LIN {X 0,Y 256.114,Z 308.577,A -85,B 0,C 180,E1 -18381.118,E2 -18381.118} C_VEL
LIN {X 0,Y 256.131,Z 308.577,A -85,B 0,C 180,E1 -18385.131,E2 -18385.131} C_VEL
LIN {X 0,Y 256.077,Z 308.586,A -85,B 0,C 180,E1 -18388.587,E2 -18388.587} C_VEL
LIN {X 0,Y 256.039,Z 308.588,A -85,B 0,C 180,E1 -18391.704,E2 -18391.704} C_VEL
LIN {X 0,Y 256.048,Z 308.59,A -85,B 0,C 180,E1 -18395.197,E2 -18395.197} C_VEL
LIN {X 0,Y 256.081,Z 308.587,A -85,B 0,C 180,E1 -18397.274,E2 -18397.274} C_VEL
LIN {X 0,Y 256.021,Z 308.597,A -85,B 0,C 180,E1 -18401.209,E2 -18401.209} C_VEL
LIN {X 0,Y 256.015,Z 308.597,A -85,B 0,C 180,E1 -18405.539,E2 -18405.539} C_VEL
LIN {X 0,Y 256.03,Z 308.591,A -85,B 0,C 180,E1 -18408.801,E2 -18408.801} C_VEL
LIN {X 0,Y 256.103,Z 308.582,A -85,B 0,C 180,E1 -18412.871,E2 -18412.871} C_VEL
LIN {X 0,Y 256.142,Z 308.689,A -85,B 0,C 180,E1 -18414.221,E2 -18414.221} C_VEL
LIN {X 0,Y 259.197,Z 322.488,A -85,B 0,C 180,E1 -18418.563,E2 -18418.563} C_VEL
LIN {X 0,Y 261.811,Z 335.171,A -85,B 0,C 180,E1 -18422.354,E2 -18422.354} C_VEL
LIN {X 0,Y 261.634,Z 338.484,A -85,B 0,C 180,E1 -18423.267,E2 -18423.267} C_VEL
LIN {X 0,Y 260.691,Z 343.829,A -85,B 0,C 180,E1 -18424.698,E2 -18424.698} C_VEL
LIN {X 0,Y 262.51,Z 368.373,A -85,B 0,C 180,E1 -18425.713,E2 -18425.713} C_VEL
LIN {X 0,Y 263.496,Z 379.827,A -85,B 0,C 180,E1 -18426.176,E2 -18426.176} C_VEL
LIN {X 0,Y 261.358,Z 445.18,A -85,B 0,C 180,E1 -18428.461,E2 -18428.461} C_VEL
LIN {X 0,Y 260.854,Z 455.2,A -85,B 0,C 180,E1 -18428.987,E2 -18428.987} C_VEL
LIN {X 0,Y 260.148,Z 464.552,A -85,B 0,C 180,E1 -18429.651,E2 -18429.651} C_VEL
LIN {X 0,Y 259.438,Z 473.095,A -85,B 0,C 180,E1 -18430.419,E2 -18430.419} C_VEL
LIN {X 0,Y 258.581,Z 483.372,A -85,B 0,C 180,E1 -18431.587,E2 -18431.587} C_VEL
LIN {X 0,Y 257.769,Z 491.491,A -85,B 0,C 180,E1 -18432.709,E2 -18432.709} C_VEL
LIN {X 0,Y 256.852,Z 500.011,A -85,B 0,C 180,E1 -18434.125,E2 -18434.125} C_VEL
LIN {X 0,Y 256.062,Z 507.913,A -85,B 0,C 180,E1 -18435.704,E2 -18435.704} C_VEL
LIN {X 0,Y 255.478,Z 514.624,A -85,B 0,C 180,E1 -18437.291,E2 -18437.291} C_VEL
LIN {X 0,Y 254.899,Z 521.569,A -85,B 0,C 180,E1 -18439.279,E2 -18439.279} C_VEL
LIN {X 0,Y 254.571,Z 527.294,A -85,B 0,C 180,E1 -18441.271,E2 -18441.271} C_VEL
LIN {X 0,Y 254.459,Z 531.171,A -85,B 0,C 180,E1 -18442.864,E2 -18442.864} C_VEL
LIN {X 0,Y 254.426,Z 535.723,A -85,B 0,C 180,E1 -18445.25,E2 -18445.25} C_VEL
LIN {X 0,Y 254.312,Z 538.017,A -85,B 0,C 180,E1 -18446.835,E2 -18446.835} C_VEL
LIN {X 0,Y 254.579,Z 541.236,A -85,B 0,C 180,E1 -18450.003,E2 -18450.003} C_VEL
LIN {X 0,Y 254.198,Z 542.076,A -85,B 0,C 180,E1 -18451.587,E2 -18451.587} C_VEL
LIN {X 0,Y 254.17,Z 542.453,A -85,B 0,C 180,E1 -18453.173,E2 -18453.173} C_VEL
LIN {X 0,Y 254.083,Z 542.355,A -85,B 0,C 180,E1 -18455.282,E2 -18455.282} C_VEL
LIN {X 0,Y 254.247,Z 541.14,A -85,B 0,C 180,E1 -18457.947,E2 -18457.947} C_VEL
LIN {X 0,Y 254.567,Z 539.931,A -85,B 0,C 180,E1 -18459.537,E2 -18459.537} C_VEL
LIN {X 0,Y 255.342,Z 537.174,A -85,B 0,C 180,E1 -18461.915,E2 -18461.915} C_VEL
LIN {X 0,Y 256.555,Z 533.388,A -85,B 0,C 180,E1 -18464.275,E2 -18464.275} C_VEL
LIN {X 0,Y 258.302,Z 528.46,A -85,B 0,C 180,E1 -18466.602,E2 -18466.602} C_VEL
LIN {X 0,Y 260.277,Z 522.255,A -85,B 0,C 180,E1 -18468.908,E2 -18468.908} C_VEL
LIN {X 0,Y 262.432,Z 515.951,A -85,B 0,C 180,E1 -18470.785,E2 -18470.785} C_VEL
LIN {X 0,Y 265.001,Z 508.371,A -85,B 0,C 180,E1 -18472.617,E2 -18472.617} C_VEL
LIN {X 0,Y 267.173,Z 501.282,A -85,B 0,C 180,E1 -18474.063,E2 -18474.063} C_VEL
LIN {X 0,Y 269.672,Z 492.854,A -85,B 0,C 180,E1 -18475.469,E2 -18475.469} C_VEL
LIN {X 0,Y 271.95,Z 484.083,A -85,B 0,C 180,E1 -18476.681,E2 -18476.681} C_VEL
LIN {X 0,Y 274.07,Z 475.043,A -85,B 0,C 180,E1 -18477.696,E2 -18477.696} C_VEL
LIN {X 0,Y 276.051,Z 464.838,A -85,B 0,C 180,E1 -18478.617,E2 -18478.617} C_VEL
LIN {X 0,Y 277.859,Z 454.072,A -85,B 0,C 180,E1 -18479.345,E2 -18479.345} C_VEL
LIN {X 0,Y 279.297,Z 443.596,A -85,B 0,C 180,E1 -18479.852,E2 -18479.852} C_VEL
LIN {X 0,Y 283.965,Z 384.409,A -85,B 0,C 180,E1 -18481.995,E2 -18481.995} C_VEL
LIN {X 0,Y 282.949,Z 372.74,A -85,B 0,C 180,E1 -18482.847,E2 -18482.847} C_VEL
LIN {X 0,Y 281.976,Z 365.365,A -85,B 0,C 180,E1 -18483.5,E2 -18483.5} C_VEL
LIN {X 0,Y 277.7,Z 356.302,A -85,B 0,C 180,E1 -18485.107,E2 -18485.107} C_VEL
LIN {X 0,Y 274.684,Z 350.616,A -85,B 0,C 180,E1 -18486.34,E2 -18486.34} C_VEL
LIN {X 0,Y 272.069,Z 346.151,A -85,B 0,C 180,E1 -18487.432,E2 -18487.432} C_VEL
LIN {X 0,Y 269.572,Z 341.715,A -85,B 0,C 180,E1 -18488.685,E2 -18488.685} C_VEL
LIN {X 0,Y 267.905,Z 336.182,A -85,B 0,C 180,E1 -18491.747,E2 -18491.747} C_VEL
LIN {X 0,Y 266.481,Z 331.991,A -85,B 0,C 180,E1 -18494.597,E2 -18494.597} C_VEL
LIN {X 0,Y 265.102,Z 328.21,A -85,B 0,C 180,E1 -18497.925,E2 -18497.925} C_VEL
LIN {X 0,Y 263.893,Z 325.058,A -85,B 0,C 180,E1 -18502.228,E2 -18502.228} C_VEL
LIN {X 0,Y 263.574,Z 324.321,A -85,B 0,C 180,E1 -18504.084,E2 -18504.084} C_VEL
LIN {X 0,Y 263.401,Z 324.098,A -85,B 0,C 180,E1 -18508.626,E2 -18508.626} C_VEL
LIN {X 0,Y 263.901,Z 324.897,A -85,B 0,C 180,E1 -18511.497,E2 -18511.497} C_VEL
LIN {X 0,Y 264.788,Z 327.071,A -85,B 0,C 180,E1 -18514.871,E2 -18514.871} C_VEL
LIN {X 0,Y 265.88,Z 329.841,A -85,B 0,C 180,E1 -18517.685,E2 -18517.685} C_VEL
LIN {X 0,Y 267.613,Z 334.155,A -85,B 0,C 180,E1 -18520.976,E2 -18520.976} C_VEL
LIN {X 0,Y 269.587,Z 339.896,A -85,B 0,C 180,E1 -18524.309,E2 -18524.309} C_VEL
LIN {X 0,Y 273.841,Z 346.836,A -85,B 0,C 180,E1 -18526.245,E2 -18526.245} C_VEL
LIN {X 0,Y 277.114,Z 352.608,A -85,B 0,C 180,E1 -18527.621,E2 -18527.621} C_VEL
LIN {X 0,Y 280.442,Z 359.089,A -85,B 0,C 180,E1 -18528.924,E2 -18528.924} C_VEL
LIN {X 0,Y 281.228,Z 361.609,A -85,B 0,C 180,E1 -18529.283,E2 -18529.283} C_VEL
LIN {X 0,Y 283.281,Z 378.778,A -85,B 0,C 180,E1 -18530.847,E2 -18530.847} C_VEL
LIN {X 0,Y 283.529,Z 382.951,A -85,B 0,C 180,E1 -18531.149,E2 -18531.149} C_VEL
LIN {X 0,Y 278.983,Z 431.266,A -85,B 0,C 180,E1 -18533.128,E2 -18533.128} C_VEL
LIN {X 0,Y 277.298,Z 444.107,A -85,B 0,C 180,E1 -18533.908,E2 -18533.908} C_VEL
LIN {X 0,Y 275.485,Z 454.611,A -85,B 0,C 180,E1 -18534.828,E2 -18534.828} C_VEL
LIN {X 0,Y 273.394,Z 464.676,A -85,B 0,C 180,E1 -18535.947,E2 -18535.947} C_VEL
LIN {X 0,Y 271.189,Z 473.801,A -85,B 0,C 180,E1 -18537.216,E2 -18537.216} C_VEL
LIN {X 0,Y 268.712,Z 482.846,A -85,B 0,C 180,E1 -18538.782,E2 -18538.782} C_VEL
LIN {X 0,Y 265.9,Z 491.692,A -85,B 0,C 180,E1 -18540.758,E2 -18540.758} C_VEL
LIN {X 0,Y 263.929,Z 497.227,A -85,B 0,C 180,E1 -18542.29,E2 -18542.29} C_VEL
LIN {X 0,Y 262.192,Z 501.907,A -85,B 0,C 180,E1 -18543.843,E2 -18543.843} C_VEL
LIN {X 0,Y 260.615,Z 505.883,A -85,B 0,C 180,E1 -18545.459,E2 -18545.459} C_VEL
LIN {X 0,Y 258.633,Z 510.251,A -85,B 0,C 180,E1 -18547.81,E2 -18547.81} C_VEL
LIN {X 0,Y 257.521,Z 512.523,A -85,B 0,C 180,E1 -18549.425,E2 -18549.425} C_VEL
LIN {X 0,Y 256.563,Z 514.125,A -85,B 0,C 180,E1 -18551.056,E2 -18551.056} C_VEL
LIN {X 0,Y 255.746,Z 515.171,A -85,B 0,C 180,E1 -18552.701,E2 -18552.701} C_VEL
LIN {X 0,Y 254.877,Z 515.787,A -85,B 0,C 180,E1 -18555.192,E2 -18555.192} C_VEL
LIN {X 0,Y 254.291,Z 515.154,A -85,B 0,C 180,E1 -18557.7,E2 -18557.7} C_VEL
LIN {X 0,Y 254.076,Z 513.537,A -85,B 0,C 180,E1 -18559.875,E2 -18559.875} C_VEL
LIN {X 0,Y 254.058,Z 511.101,A -85,B 0,C 180,E1 -18561.93,E2 -18561.93} C_VEL
LIN {X 0,Y 254.346,Z 506.669,A -85,B 0,C 180,E1 -18564.487,E2 -18564.487} C_VEL
LIN {X 0,Y 254.594,Z 502.794,A -85,B 0,C 180,E1 -18566.212,E2 -18566.212} C_VEL
LIN {X 0,Y 255.028,Z 497.402,A -85,B 0,C 180,E1 -18568.138,E2 -18568.138} C_VEL
LIN {X 0,Y 255.458,Z 492.196,A -85,B 0,C 180,E1 -18569.684,E2 -18569.684} C_VEL
LIN {X 0,Y 256.07,Z 485.08,A -85,B 0,C 180,E1 -18571.432,E2 -18571.432} C_VEL
LIN {X 0,Y 256.763,Z 477.44,A -85,B 0,C 180,E1 -18572.983,E2 -18572.983} C_VEL
LIN {X 0,Y 257.589,Z 468.46,A -85,B 0,C 180,E1 -18574.482,E2 -18574.482} C_VEL
LIN {X 0,Y 258.507,Z 457.069,A -85,B 0,C 180,E1 -18576.003,E2 -18576.003} C_VEL
LIN {X 0,Y 259.295,Z 446.195,A -85,B 0,C 180,E1 -18577.091,E2 -18577.091} C_VEL
LIN {X 0,Y 259.852,Z 435.418,A -85,B 0,C 180,E1 -18577.913,E2 -18577.913} C_VEL
LIN {X 0,Y 260.388,Z 424.12,A -85,B 0,C 180,E1 -18578.524,E2 -18578.524} C_VEL
LIN {X 0,Y 262.234,Z 371.857,A -85,B 0,C 180,E1 -18580.561,E2 -18580.561} C_VEL
LIN {X 0,Y 258.762,Z 340.403,A -85,B 0,C 180,E1 -18582.011,E2 -18582.011} C_VEL
LIN {X 0,Y 260.138,Z 329.508,A -85,B 0,C 180,E1 -18585.379,E2 -18585.379} C_VEL
LIN {X 0,Y 258.66,Z 320.931,A -85,B 0,C 180,E1 -18588.266,E2 -18588.266} C_VEL
LIN {X 0,Y 256.154,Z 308.576,A -85,B 0,C 180,E1 -18592.672,E2 -18592.672} C_VEL
LIN {X 0,Y 256.068,Z 308.585,A -85,B 0,C 180,E1 -18596.707,E2 -18596.707} C_VEL
LIN {X 0,Y 256.044,Z 308.591,A -85,B 0,C 180,E1 -18600.391,E2 -18600.391} C_VEL
LIN {X 0,Y 256.069,Z 308.588,A -85,B 0,C 180,E1 -18603.951,E2 -18603.951} C_VEL
LIN {X 0,Y 256.062,Z 308.586,A -85,B 0,C 180,E1 -18607.402,E2 -18607.402} C_VEL
LIN {X 0,Y 256.134,Z 308.581,A -85,B 0,C 180,E1 -18610.774,E2 -18610.774} C_VEL
LIN {X 0,Y 256.236,Z 308.564,A -85,B 0,C 180,E1 -18614.079,E2 -18614.079} C_VEL
LIN {X 0,Y 256.293,Z 308.56,A -85,B 0,C 180,E1 -18618.931,E2 -18618.931} C_VEL
LIN {X 0,Y 256.473,Z 308.534,A -85,B 0,C 180,E1 -18622.123,E2 -18622.123} C_VEL
LIN {X 0,Y 256.447,Z 308.537,A -85,B 0,C 180,E1 -18626.855,E2 -18626.855} C_VEL
LIN {X 0,Y 256.698,Z 308.507,A -85,B 0,C 180,E1 -18628.428,E2 -18628.428} C_VEL
LIN {X 0,Y 256.697,Z 308.509,A -85,B 0,C 180,E1 -18631.566,E2 -18631.566} C_VEL
LIN {X 0,Y 256.455,Z 308.54,A -85,B 0,C 180,E1 -18636.289,E2 -18636.289} C_VEL
LIN {X 0,Y 256.428,Z 308.54,A -85,B 0,C 180,E1 -18639.461,E2 -18639.461} C_VEL
LIN {X 0,Y 256.231,Z 308.566,A -85,B 0,C 180,E1 -18644.287,E2 -18644.287} C_VEL
LIN {X 0,Y 256.16,Z 308.574,A -85,B 0,C 180,E1 -18647.56,E2 -18647.56} C_VEL
LIN {X 0,Y 256.117,Z 308.58,A -85,B 0,C 180,E1 -18651.093,E2 -18651.093} C_VEL
LIN {X 0,Y 256.125,Z 308.582,A -85,B 0,C 180,E1 -18655.106,E2 -18655.106} C_VEL
LIN {X 0,Y 256.042,Z 308.589,A -85,B 0,C 180,E1 -18659.602,E2 -18659.602} C_VEL
LIN {X 0,Y 256.053,Z 308.588,A -85,B 0,C 180,E1 -18663.287,E2 -18663.287} C_VEL
LIN {X 0,Y 256.095,Z 308.582,A -85,B 0,C 180,E1 -18667.263,E2 -18667.263} C_VEL
LIN {X 0,Y 256.035,Z 308.588,A -85,B 0,C 180,E1 -18671.198,E2 -18671.198} C_VEL
LIN {X 0,Y 256.019,Z 308.591,A -85,B 0,C 180,E1 -18675.529,E2 -18675.529} C_VEL
LIN {X 0,Y 256.026,Z 308.592,A -85,B 0,C 180,E1 -18678.79,E2 -18678.79} C_VEL
LIN {X 0,Y 256.099,Z 308.585,A -85,B 0,C 180,E1 -18682.861,E2 -18682.861} C_VEL
LIN {X 0,Y 256.039,Z 308.59,A -85,B 0,C 180,E1 -18686.702,E2 -18686.702} C_VEL
LIN {X 0,Y 256.082,Z 308.583,A -85,B 0,C 180,E1 -18690.395,E2 -18690.395} C_VEL
LIN {X 0,Y 256.136,Z 308.576,A -85,B 0,C 180,E1 -18694.867,E2 -18694.867} C_VEL
LIN {X 0,Y 256.087,Z 308.583,A -85,B 0,C 180,E1 -18699.097,E2 -18699.097} C_VEL
LIN {X 0,Y 256.19,Z 308.572,A -85,B 0,C 180,E1 -18704.077,E2 -18704.077} C_VEL
LIN {X 0,Y 256.251,Z 308.563,A -85,B 0,C 180,E1 -18708.931,E2 -18708.931} C_VEL
LIN {X 0,Y 256.469,Z 308.537,A -85,B 0,C 180,E1 -18712.124,E2 -18712.124} C_VEL
LIN {X 0,Y 256.464,Z 308.54,A -85,B 0,C 180,E1 -18716.857,E2 -18716.857} C_VEL
LIN {X 0,Y 256.713,Z 308.504,A -85,B 0,C 180,E1 -18719.999,E2 -18719.999} C_VEL
LIN {X 0,Y 256.453,Z 308.54,A -85,B 0,C 180,E1 -18723.141,E2 -18723.141} C_VEL
LIN {X 0,Y 256.468,Z 308.536,A -85,B 0,C 180,E1 -18727.874,E2 -18727.874} C_VEL
LIN {X 0,Y 256.233,Z 308.563,A -85,B 0,C 180,E1 -18731.3,E2 -18731.3} C_VEL
LIN {X 0,Y 256.224,Z 308.57,A -85,B 0,C 180,E1 -18735.919,E2 -18735.919} C_VEL
LIN {X 0,Y 256.128,Z 308.576,A -85,B 0,C 180,E1 -18738.13,E2 -18738.13} C_VEL
LIN {X 0,Y 255.453,Z 308.663,A -85,B 0,C 180,E1 -18739.44,E2 -18739.44} C_VEL
LIN {X 0,Y 252.641,Z 309.011,A -85,B 0,C 180,E1 -18741.579,E2 -18741.579} C_VEL
LIN {X 0,Y 250.245,Z 309.312,A -85,B 0,C 180,E1 -18743.318,E2 -18743.318} C_VEL
LIN {X 0,Y 249.191,Z 309.444,A -85,B 0,C 180,E1 -18744.666,E2 -18744.666} C_VEL
LIN {X 0,Y 249.091,Z 309.454,A -85,B 0,C 180,E1 -18745.123,E2 -18745.123} C_VEL
LIN {X 0,Y 249.019,Z 309.462,A -85,B 0,C 180,E1 -18748.983,E2 -18748.983} C_VEL
LIN {X 0,Y 248.994,Z 309.468,A -85,B 0,C 180,E1 -18752.43,E2 -18752.43} C_VEL
LIN {X 0,Y 248.996,Z 309.466,A -85,B 0,C 180,E1 -18756.35,E2 -18756.35} C_VEL
LIN {X 0,Y 248.961,Z 309.472,A -85,B 0,C 180,E1 -18760.486,E2 -18760.486} C_VEL
LIN {X 0,Y 248.97,Z 309.471,A -85,B 0,C 180,E1 -18762.794,E2 -18762.794} C_VEL
LIN {X 0,Y 248.984,Z 309.471,A -85,B 0,C 180,E1 -18767.366,E2 -18767.366} C_VEL
LIN {X 0,Y 249.002,Z 309.47,A -85,B 0,C 180,E1 -18771.624,E2 -18771.624} C_VEL
LIN {X 0,Y 249.091,Z 309.561,A -85,B 0,C 180,E1 -18773.797,E2 -18773.797} C_VEL
LIN {X 0,Y 252.249,Z 323.917,A -85,B 0,C 180,E1 -18778.434,E2 -18778.434} C_VEL
LIN {X 0,Y 254.682,Z 335.639,A -85,B 0,C 180,E1 -18782.03,E2 -18782.03} C_VEL
LIN {X 0,Y 254.729,Z 338.753,A -85,B 0,C 180,E1 -18782.926,E2 -18782.926} C_VEL
LIN {X 0,Y 253.753,Z 344.225,A -85,B 0,C 180,E1 -18784.369,E2 -18784.369} C_VEL
LIN {X 0,Y 255.793,Z 371.229,A -85,B 0,C 180,E1 -18785.501,E2 -18785.501} C_VEL
LIN {X 0,Y 256.565,Z 379.574,A -85,B 0,C 180,E1 -18785.853,E2 -18785.853} C_VEL
LIN {X 0,Y 254.365,Z 444.942,A -85,B 0,C 180,E1 -18788.212,E2 -18788.212} C_VEL
LIN {X 0,Y 253.843,Z 454.922,A -85,B 0,C 180,E1 -18788.751,E2 -18788.751} C_VEL
LIN {X 0,Y 253.09,Z 464.842,A -85,B 0,C 180,E1 -18789.483,E2 -18789.483} C_VEL
LIN {X 0,Y 252.375,Z 473.258,A -85,B 0,C 180,E1 -18790.272,E2 -18790.272} C_VEL
LIN {X 0,Y 251.502,Z 483.435,A -85,B 0,C 180,E1 -18791.472,E2 -18791.472} C_VEL
LIN {X 0,Y 250.668,Z 491.507,A -85,B 0,C 180,E1 -18792.627,E2 -18792.627} C_VEL
LIN {X 0,Y 249.746,Z 499.952,A -85,B 0,C 180,E1 -18794.081,E2 -18794.081} C_VEL
LIN {X 0,Y 248.973,Z 507.813,A -85,B 0,C 180,E1 -18795.705,E2 -18795.705} C_VEL
LIN {X 0,Y 248.37,Z 514.477,A -85,B 0,C 180,E1 -18797.337,E2 -18797.337} C_VEL
LIN {X 0,Y 247.802,Z 521.386,A -85,B 0,C 180,E1 -18799.381,E2 -18799.381} C_VEL
LIN {X 0,Y 247.534,Z 526.093,A -85,B 0,C 180,E1 -18801.02,E2 -18801.02} C_VEL
LIN {X 0,Y 247.369,Z 531.706,A -85,B 0,C 180,E1 -18803.479,E2 -18803.479} C_VEL
LIN {X 0,Y 247.376,Z 534.77,A -85,B 0,C 180,E1 -18805.115,E2 -18805.115} C_VEL
LIN {X 0,Y 247.282,Z 539.046,A -85,B 0,C 180,E1 -18808.375,E2 -18808.375} C_VEL
LIN {X 0,Y 247.524,Z 540.587,A -85,B 0,C 180,E1 -18810.003,E2 -18810.003} C_VEL
LIN {X 0,Y 247.097,Z 541.956,A -85,B 0,C 180,E1 -18813.264,E2 -18813.264} C_VEL
LIN {X 0,Y 246.987,Z 542.064,A -85,B 0,C 180,E1 -18815.185,E2 -18815.185} C_VEL
LIN {X 0,Y 247.186,Z 540.907,A -85,B 0,C 180,E1 -18818.175,E2 -18818.175} C_VEL
LIN {X 0,Y 247.546,Z 539.777,A -85,B 0,C 180,E1 -18819.81,E2 -18819.81} C_VEL
LIN {X 0,Y 248.355,Z 537.18,A -85,B 0,C 180,E1 -18822.256,E2 -18822.256} C_VEL
LIN {X 0,Y 249.684,Z 533.567,A -85,B 0,C 180,E1 -18824.676,E2 -18824.676} C_VEL
LIN {X 0,Y 251.515,Z 528.837,A -85,B 0,C 180,E1 -18827.063,E2 -18827.063} C_VEL
LIN {X 0,Y 253.59,Z 522.856,A -85,B 0,C 180,E1 -18829.426,E2 -18829.426} C_VEL
LIN {X 0,Y 256.338,Z 515.399,A -85,B 0,C 180,E1 -18831.725,E2 -18831.725} C_VEL
LIN {X 0,Y 259.098,Z 507.837,A -85,B 0,C 180,E1 -18833.585,E2 -18833.585} C_VEL
LIN {X 0,Y 261.414,Z 500.71,A -85,B 0,C 180,E1 -18835.052,E2 -18835.052} C_VEL
LIN {X 0,Y 264.071,Z 492.227,A -85,B 0,C 180,E1 -18836.474,E2 -18836.474} C_VEL
LIN {X 0,Y 266.497,Z 483.453,A -85,B 0,C 180,E1 -18837.698,E2 -18837.698} C_VEL
LIN {X 0,Y 268.708,Z 474.488,A -85,B 0,C 180,E1 -18838.725,E2 -18838.725} C_VEL
LIN {X 0,Y 270.801,Z 464.384,A -85,B 0,C 180,E1 -18839.652,E2 -18839.652} C_VEL
LIN {X 0,Y 272.745,Z 453.678,A -85,B 0,C 180,E1 -18840.377,E2 -18840.377} C_VEL
LIN {X 0,Y 274.212,Z 443.294,A -85,B 0,C 180,E1 -18840.887,E2 -18840.887} C_VEL
LIN {X 0,Y 279.082,Z 385.56,A -85,B 0,C 180,E1 -18843.024,E2 -18843.024} C_VEL
LIN {X 0,Y 278.145,Z 373.444,A -85,B 0,C 180,E1 -18843.959,E2 -18843.959} C_VEL
LIN {X 0,Y 277.492,Z 369.039,A -85,B 0,C 180,E1 -18844.387,E2 -18844.387} C_VEL
LIN {X 0,Y 273.757,Z 360.823,A -85,B 0,C 180,E1 -18845.922,E2 -18845.922} C_VEL
LIN {X 0,Y 271.155,Z 355.812,A -85,B 0,C 180,E1 -18847.037,E2 -18847.037} C_VEL
LIN {X 0,Y 268.946,Z 351.819,A -85,B 0,C 180,E1 -18848.051,E2 -18848.051} C_VEL
LIN {X 0,Y 265.932,Z 346.837,A -85,B 0,C 180,E1 -18849.507,E2 -18849.507} C_VEL
LIN {X 0,Y 262.807,Z 341.689,A -85,B 0,C 180,E1 -18851.279,E2 -18851.279} C_VEL
LIN {X 0,Y 261.347,Z 337.153,A -85,B 0,C 180,E1 -18854.36,E2 -18854.36} C_VEL
LIN {X 0,Y 260.116,Z 333.559,A -85,B 0,C 180,E1 -18857.511,E2 -18857.511} C_VEL
LIN {X 0,Y 258.911,Z 330.251,A -85,B 0,C 180,E1 -18861.921,E2 -18861.921} C_VEL
LIN {X 0,Y 258.743,Z 329.583,A -85,B 0,C 180,E1 -18863.305,E2 -18863.305} C_VEL
LIN {X 0,Y 258.326,Z 329.063,A -85,B 0,C 180,E1 -18867.496,E2 -18867.496} C_VEL
LIN {X 0,Y 258.727,Z 329.674,A -85,B 0,C 180,E1 -18870.73,E2 -18870.73} C_VEL
LIN {X 0,Y 259.348,Z 331.015,A -85,B 0,C 180,E1 -18873.409,E2 -18873.409} C_VEL
LIN {X 0,Y 260.395,Z 333.627,A -85,B 0,C 180,E1 -18876.58,E2 -18876.58} C_VEL
LIN {X 0,Y 261.852,Z 337.573,A -85,B 0,C 180,E1 -18879.942,E2 -18879.942} C_VEL
LIN {X 0,Y 262.835,Z 340.258,A -85,B 0,C 180,E1 -18881.692,E2 -18881.692} C_VEL
LIN {X 0,Y 267.268,Z 346.965,A -85,B 0,C 180,E1 -18884.071,E2 -18884.071} C_VEL
LIN {X 0,Y 270.636,Z 352.656,A -85,B 0,C 180,E1 -18885.703,E2 -18885.703} C_VEL
LIN {X 0,Y 274.341,Z 359.4,A -85,B 0,C 180,E1 -18887.318,E2 -18887.318} C_VEL
LIN {X 0,Y 276.669,Z 364.494,A -85,B 0,C 180,E1 -18888.326,E2 -18888.326} C_VEL
LIN {X 0,Y 278.512,Z 381.03,A -85,B 0,C 180,E1 -18889.884,E2 -18889.884} C_VEL
LIN {X 0,Y 278.564,Z 385.068,A -85,B 0,C 180,E1 -18890.159,E2 -18890.159} C_VEL
LIN {X 0,Y 273.873,Z 431.859,A -85,B 0,C 180,E1 -18892.119,E2 -18892.119} C_VEL
LIN {X 0,Y 272.197,Z 444.046,A -85,B 0,C 180,E1 -18892.863,E2 -18892.863} C_VEL
LIN {X 0,Y 270.197,Z 455.143,A -85,B 0,C 180,E1 -18893.841,E2 -18893.841} C_VEL
LIN {X 0,Y 268.114,Z 464.536,A -85,B 0,C 180,E1 -18894.897,E2 -18894.897} C_VEL
LIN {X 0,Y 266.027,Z 472.669,A -85,B 0,C 180,E1 -18896.024,E2 -18896.024} C_VEL
LIN {X 0,Y 263.793,Z 480.394,A -85,B 0,C 180,E1 -18897.329,E2 -18897.329} C_VEL
LIN {X 0,Y 261.635,Z 487.24,A -85,B 0,C 180,E1 -18898.714,E2 -18898.714} C_VEL
LIN {X 0,Y 259.753,Z 492.621,A -85,B 0,C 180,E1 -18900.001,E2 -18900.001} C_VEL
LIN {X 0,Y 257.69,Z 498.08,A -85,B 0,C 180,E1 -18901.564,E2 -18901.564} C_VEL
LIN {X 0,Y 255.803,Z 502.673,A -85,B 0,C 180,E1 -18903.151,E2 -18903.151} C_VEL
LIN {X 0,Y 253.946,Z 506.877,A -85,B 0,C 180,E1 -18904.955,E2 -18904.955} C_VEL
LIN {X 0,Y 251.991,Z 510.864,A -85,B 0,C 180,E1 -18907.211,E2 -18907.211} C_VEL
LIN {X 0,Y 249.934,Z 514.392,A -85,B 0,C 180,E1 -18910.218,E2 -18910.218} C_VEL
LIN {X 0,Y 248.487,Z 516.075,A -85,B 0,C 180,E1 -18913.078,E2 -18913.078} C_VEL
LIN {X 0,Y 247.749,Z 516.239,A -85,B 0,C 180,E1 -18915.323,E2 -18915.323} C_VEL
LIN {X 0,Y 247.117,Z 514.966,A -85,B 0,C 180,E1 -18918.231,E2 -18918.231} C_VEL
LIN {X 0,Y 246.984,Z 513.334,A -85,B 0,C 180,E1 -18920.118,E2 -18920.118} C_VEL
LIN {X 0,Y 246.97,Z 511.441,A -85,B 0,C 180,E1 -18921.713,E2 -18921.713} C_VEL
LIN {X 0,Y 247.197,Z 507.641,A -85,B 0,C 180,E1 -18924.012,E2 -18924.012} C_VEL
LIN {X 0,Y 247.494,Z 503.075,A -85,B 0,C 180,E1 -18926.114,E2 -18926.114} C_VEL
LIN {X 0,Y 247.937,Z 497.45,A -85,B 0,C 180,E1 -18928.169,E2 -18928.169} C_VEL
LIN {X 0,Y 248.35,Z 492.473,A -85,B 0,C 180,E1 -18929.686,E2 -18929.686} C_VEL
LIN {X 0,Y 248.987,Z 485.365,A -85,B 0,C 180,E1 -18931.48,E2 -18931.48} C_VEL
LIN {X 0,Y 249.684,Z 477.834,A -85,B 0,C 180,E1 -18933.05,E2 -18933.05} C_VEL
LIN {X 0,Y 250.379,Z 470.095,A -85,B 0,C 180,E1 -18934.396,E2 -18934.396} C_VEL
LIN {X 0,Y 251.048,Z 462.425,A -85,B 0,C 180,E1 -18935.514,E2 -18935.514} C_VEL
LIN {X 0,Y 251.709,Z 453.018,A -85,B 0,C 180,E1 -18936.643,E2 -18936.643} C_VEL
LIN {X 0,Y 252.518,Z 442.541,A -85,B 0,C 180,E1 -18937.631,E2 -18937.631} C_VEL
LIN {X 0,Y 253.17,Z 429.531,A -85,B 0,C 180,E1 -18938.511,E2 -18938.511} C_VEL
LIN {X 0,Y 254.256,Z 400.469,A -85,B 0,C 180,E1 -18939.734,E2 -18939.734} C_VEL
LIN {X 0,Y 255.242,Z 372.305,A -85,B 0,C 180,E1 -18940.859,E2 -18940.859} C_VEL
LIN {X 0,Y 251.813,Z 340.434,A -85,B 0,C 180,E1 -18942.391,E2 -18942.391} C_VEL
LIN {X 0,Y 253.127,Z 330.314,A -85,B 0,C 180,E1 -18945.595,E2 -18945.595} C_VEL
LIN {X 0,Y 251.53,Z 321.534,A -85,B 0,C 180,E1 -18948.63,E2 -18948.63} C_VEL
LIN {X 0,Y 249.184,Z 310,A -85,B 0,C 180,E1 -18952.816,E2 -18952.816} C_VEL
LIN {X 0,Y 249.098,Z 309.455,A -85,B 0,C 180,E1 -18953.127,E2 -18953.127} C_VEL
LIN {X 0,Y 249.034,Z 309.465,A -85,B 0,C 180,E1 -18957.849,E2 -18957.849} C_VEL
LIN {X 0,Y 249.038,Z 309.462,A -85,B 0,C 180,E1 -18961.33,E2 -18961.33} C_VEL
LIN {X 0,Y 249.059,Z 309.459,A -85,B 0,C 180,E1 -18964.958,E2 -18964.958} C_VEL
LIN {X 0,Y 249.056,Z 309.463,A -85,B 0,C 180,E1 -18968.627,E2 -18968.627} C_VEL
LIN {X 0,Y 249.164,Z 309.445,A -85,B 0,C 180,E1 -18973.615,E2 -18973.615} C_VEL
LIN {X 0,Y 249.192,Z 309.444,A -85,B 0,C 180,E1 -18976.958,E2 -18976.958} C_VEL
LIN {X 0,Y 249.389,Z 309.418,A -85,B 0,C 180,E1 -18980.52,E2 -18980.52} C_VEL
LIN {X 0,Y 249.43,Z 309.414,A -85,B 0,C 180,E1 -18983.526,E2 -18983.526} C_VEL
LIN {X 0,Y 249.659,Z 309.384,A -85,B 0,C 180,E1 -18988.384,E2 -18988.384} C_VEL
LIN {X 0,Y 249.658,Z 309.387,A -85,B 0,C 180,E1 -18991.61,E2 -18991.61} C_VEL
LIN {X 0,Y 249.429,Z 309.414,A -85,B 0,C 180,E1 -18996.467,E2 -18996.467} C_VEL
LIN {X 0,Y 249.345,Z 309.424,A -85,B 0,C 180,E1 -18999.732,E2 -18999.732} C_VEL
LIN {X 0,Y 249.17,Z 309.448,A -85,B 0,C 180,E1 -19004.701,E2 -19004.701} C_VEL
LIN {X 0,Y 249.092,Z 309.455,A -85,B 0,C 180,E1 -19008.076,E2 -19008.076} C_VEL
LIN {X 0,Y 249.041,Z 309.459,A -85,B 0,C 180,E1 -19011.517,E2 -19011.517} C_VEL
LIN {X 0,Y 249.077,Z 309.459,A -85,B 0,C 180,E1 -19015.454,E2 -19015.454} C_VEL
LIN {X 0,Y 249.025,Z 309.464,A -85,B 0,C 180,E1 -19018.967,E2 -19018.967} C_VEL
LIN {X 0,Y 249.015,Z 309.463,A -85,B 0,C 180,E1 -19022.421,E2 -19022.421} C_VEL
LIN {X 0,Y 249.012,Z 309.465,A -85,B 0,C 180,E1 -19026.34,E2 -19026.34} C_VEL
LIN {X 0,Y 248.974,Z 309.469,A -85,B 0,C 180,E1 -19030.475,E2 -19030.475} C_VEL
LIN {X 0,Y 248.982,Z 309.469,A -85,B 0,C 180,E1 -19032.784,E2 -19032.784} C_VEL
LIN {X 0,Y 248.984,Z 309.466,A -85,B 0,C 180,E1 -19037.355,E2 -19037.355} C_VEL
LIN {X 0,Y 249.015,Z 309.465,A -85,B 0,C 180,E1 -19042.196,E2 -19042.196} C_VEL
LIN {X 0,Y 249.015,Z 309.463,A -85,B 0,C 180,E1 -19045.634,E2 -19045.634} C_VEL
LIN {X 0,Y 249.021,Z 309.465,A -85,B 0,C 180,E1 -19049.468,E2 -19049.468} C_VEL
LIN {X 0,Y 249.037,Z 309.464,A -85,B 0,C 180,E1 -19053.157,E2 -19053.157} C_VEL
LIN {X 0,Y 249.022,Z 309.46,A -85,B 0,C 180,E1 -19056.726,E2 -19056.726} C_VEL
LIN {X 0,Y 249.009,Z 309.466,A -85,B 0,C 180,E1 -19060.202,E2 -19060.202} C_VEL
LIN {X 0,Y 249.122,Z 309.452,A -85,B 0,C 180,E1 -19063.613,E2 -19063.613} C_VEL
LIN {X 0,Y 249.194,Z 309.443,A -85,B 0,C 180,E1 -19068.613,E2 -19068.613} C_VEL
LIN {X 0,Y 249.407,Z 309.416,A -85,B 0,C 180,E1 -19071.9,E2 -19071.9} C_VEL
LIN {X 0,Y 249.257,Z 309.434,A -85,B 0,C 180,E1 -19075.147,E2 -19075.147} C_VEL
LIN {X 0,Y 249.636,Z 309.388,A -85,B 0,C 180,E1 -19078.386,E2 -19078.386} C_VEL
LIN {X 0,Y 249.632,Z 309.386,A -85,B 0,C 180,E1 -19081.612,E2 -19081.612} C_VEL
LIN {X 0,Y 249.407,Z 309.415,A -85,B 0,C 180,E1 -19086.471,E2 -19086.471} C_VEL
LIN {X 0,Y 249.304,Z 309.429,A -85,B 0,C 180,E1 -19089.737,E2 -19089.737} C_VEL
LIN {X 0,Y 249.145,Z 309.447,A -85,B 0,C 180,E1 -19094.706,E2 -19094.706} C_VEL
LIN {X 0,Y 249.089,Z 309.457,A -85,B 0,C 180,E1 -19098.102,E2 -19098.102} C_VEL
LIN {X 0,Y 249.047,Z 309.458,A -85,B 0,C 180,E1 -19101.521,E2 -19101.521} C_VEL
LIN {X 0,Y 249.091,Z 309.454,A -85,B 0,C 180,E1 -19105.123,E2 -19105.123} C_VEL
LIN {X 0,Y 248.364,Z 309.549,A -85,B 0,C 180,E1 -19106.472,E2 -19106.472} C_VEL
LIN {X 0,Y 245.434,Z 309.911,A -85,B 0,C 180,E1 -19108.67,E2 -19108.67} C_VEL
LIN {X 0,Y 243,Z 310.213,A -85,B 0,C 180,E1 -19110.46,E2 -19110.46} C_VEL
LIN {X 0,Y 241.997,Z 310.337,A -85,B 0,C 180,E1 -19111.85,E2 -19111.85} C_VEL
LIN {X 0,Y 241.937,Z 310.346,A -85,B 0,C 180,E1 -19112.321,E2 -19112.321} C_VEL
LIN {X 0,Y 241.948,Z 310.344,A -85,B 0,C 180,E1 -19115.591,E2 -19115.591} C_VEL
LIN {X 0,Y 241.917,Z 310.35,A -85,B 0,C 180,E1 -19119.726,E2 -19119.726} C_VEL
LIN {X 0,Y 241.891,Z 310.352,A -85,B 0,C 180,E1 -19124.21,E2 -19124.21} C_VEL
LIN {X 0,Y 241.909,Z 310.352,A -85,B 0,C 180,E1 -19128.081,E2 -19128.081} C_VEL
LIN {X 0,Y 241.974,Z 310.344,A -85,B 0,C 180,E1 -19132.424,E2 -19132.424} C_VEL
LIN {X 0,Y 242.042,Z 310.45,A -85,B 0,C 180,E1 -19133.357,E2 -19133.357} C_VEL
LIN {X 0,Y 244.685,Z 322.589,A -85,B 0,C 180,E1 -19137.423,E2 -19137.423} C_VEL
LIN {X 0,Y 247.169,Z 334.123,A -85,B 0,C 180,E1 -19141.101,E2 -19141.101} C_VEL
LIN {X 0,Y 247.801,Z 337.695,A -85,B 0,C 180,E1 -19142.201,E2 -19142.201} C_VEL
LIN {X 0,Y 247.244,Z 341.902,A -85,B 0,C 180,E1 -19143.41,E2 -19143.41} C_VEL
LIN {X 0,Y 246.837,Z 344.096,A -85,B 0,C 180,E1 -19143.989,E2 -19143.989} C_VEL
LIN {X 0,Y 248.625,Z 369.376,A -85,B 0,C 180,E1 -19145.074,E2 -19145.074} C_VEL
LIN {X 0,Y 249.577,Z 380.376,A -85,B 0,C 180,E1 -19145.549,E2 -19145.549} C_VEL
LIN {X 0,Y 247.389,Z 444.693,A -85,B 0,C 180,E1 -19147.949,E2 -19147.949} C_VEL
LIN {X 0,Y 246.846,Z 454.629,A -85,B 0,C 180,E1 -19148.502,E2 -19148.502} C_VEL
LIN {X 0,Y 246.127,Z 463.928,A -85,B 0,C 180,E1 -19149.203,E2 -19149.203} C_VEL
LIN {X 0,Y 245.323,Z 473.354,A -85,B 0,C 180,E1 -19150.117,E2 -19150.117} C_VEL
LIN {X 0,Y 244.558,Z 481.929,A -85,B 0,C 180,E1 -19151.143,E2 -19151.143} C_VEL
LIN {X 0,Y 243.637,Z 491.002,A -85,B 0,C 180,E1 -19152.469,E2 -19152.469} C_VEL
LIN {X 0,Y 242.66,Z 499.803,A -85,B 0,C 180,E1 -19154.035,E2 -19154.035} C_VEL
LIN {X 0,Y 241.87,Z 507.61,A -85,B 0,C 180,E1 -19155.706,E2 -19155.706} C_VEL
LIN {X 0,Y 241.291,Z 514.24,A -85,B 0,C 180,E1 -19157.387,E2 -19157.387} C_VEL
LIN {X 0,Y 240.735,Z 521.11,A -85,B 0,C 180,E1 -19159.491,E2 -19159.491} C_VEL
LIN {X 0,Y 240.41,Z 526.758,A -85,B 0,C 180,E1 -19161.599,E2 -19161.599} C_VEL
LIN {X 0,Y 240.315,Z 531.694,A -85,B 0,C 180,E1 -19163.887,E2 -19163.887} C_VEL
LIN {X 0,Y 240.26,Z 535.039,A -85,B 0,C 180,E1 -19165.81,E2 -19165.81} C_VEL
LIN {X 0,Y 240.21,Z 538.263,A -85,B 0,C 180,E1 -19168.327,E2 -19168.327} C_VEL
LIN {X 0,Y 240.469,Z 539.844,A -85,B 0,C 180,E1 -19170.003,E2 -19170.003} C_VEL
LIN {X 0,Y 240.026,Z 541.459,A -85,B 0,C 180,E1 -19173.36,E2 -19173.36} C_VEL
LIN {X 0,Y 239.909,Z 541.634,A -85,B 0,C 180,E1 -19175.13,E2 -19175.13} C_VEL
LIN {X 0,Y 240.145,Z 540.7,A -85,B 0,C 180,E1 -19178.417,E2 -19178.417} C_VEL
LIN {X 0,Y 240.511,Z 539.572,A -85,B 0,C 180,E1 -19180.1,E2 -19180.1} C_VEL
LIN {X 0,Y 241.756,Z 536.13,A -85,B 0,C 180,E1 -19183.45,E2 -19183.45} C_VEL
LIN {X 0,Y 243.427,Z 532.311,A -85,B 0,C 180,E1 -19185.921,E2 -19185.921} C_VEL
LIN {X 0,Y 245.446,Z 527.384,A -85,B 0,C 180,E1 -19188.361,E2 -19188.361} C_VEL
LIN {X 0,Y 247.784,Z 521.421,A -85,B 0,C 180,E1 -19190.68,E2 -19190.68} C_VEL
LIN {X 0,Y 250.362,Z 514.89,A -85,B 0,C 180,E1 -19192.706,E2 -19192.706} C_VEL
LIN {X 0,Y 253.236,Z 507.32,A -85,B 0,C 180,E1 -19194.602,E2 -19194.602} C_VEL
LIN {X 0,Y 255.78,Z 500.237,A -85,B 0,C 180,E1 -19196.081,E2 -19196.081} C_VEL
LIN {X 0,Y 258.579,Z 491.84,A -85,B 0,C 180,E1 -19197.52,E2 -19197.52} C_VEL
LIN {X 0,Y 261.132,Z 483.11,A -85,B 0,C 180,E1 -19198.756,E2 -19198.756} C_VEL
LIN {X 0,Y 263.459,Z 474.138,A -85,B 0,C 180,E1 -19199.791,E2 -19199.791} C_VEL
LIN {X 0,Y 265.696,Z 464.005,A -85,B 0,C 180,E1 -19200.72,E2 -19200.72} C_VEL
LIN {X 0,Y 267.716,Z 453.345,A -85,B 0,C 180,E1 -19201.45,E2 -19201.45} C_VEL
LIN {X 0,Y 269.262,Z 443.113,A -85,B 0,C 180,E1 -19201.962,E2 -19201.962} C_VEL
LIN {X 0,Y 274.383,Z 386.982,A -85,B 0,C 180,E1 -19204.085,E2 -19204.085} C_VEL
LIN {X 0,Y 273.543,Z 375.524,A -85,B 0,C 180,E1 -19205.012,E2 -19205.012} C_VEL
LIN {X 0,Y 273.158,Z 372.747,A -85,B 0,C 180,E1 -19205.301,E2 -19205.301} C_VEL
LIN {X 0,Y 269.928,Z 365.493,A -85,B 0,C 180,E1 -19206.734,E2 -19206.734} C_VEL
LIN {X 0,Y 266.484,Z 358.478,A -85,B 0,C 180,E1 -19208.382,E2 -19208.382} C_VEL
LIN {X 0,Y 262.9,Z 352.452,A -85,B 0,C 180,E1 -19210.212,E2 -19210.212} C_VEL
LIN {X 0,Y 259.689,Z 347.231,A -85,B 0,C 180,E1 -19212.09,E2 -19212.09} C_VEL
LIN {X 0,Y 255.94,Z 341.51,A -85,B 0,C 180,E1 -19214.763,E2 -19214.763} C_VEL
LIN {X 0,Y 254.724,Z 337.927,A -85,B 0,C 180,E1 -19218.153,E2 -19218.153} C_VEL
LIN {X 0,Y 253.801,Z 335.016,A -85,B 0,C 180,E1 -19222.469,E2 -19222.469} C_VEL
LIN {X 0,Y 253.525,Z 334.347,A -85,B 0,C 180,E1 -19224.4,E2 -19224.4} C_VEL
LIN {X 0,Y 253.477,Z 334.338,A -85,B 0,C 180,E1 -19229.259,E2 -19229.259} C_VEL
LIN {X 0,Y 254.037,Z 335.373,A -85,B 0,C 180,E1 -19232.283,E2 -19232.283} C_VEL
LIN {X 0,Y 254.883,Z 337.721,A -85,B 0,C 180,E1 -19235.57,E2 -19235.57} C_VEL
LIN {X 0,Y 255.994,Z 340.539,A -85,B 0,C 180,E1 -19238.246,E2 -19238.246} C_VEL
LIN {X 0,Y 260.594,Z 346.995,A -85,B 0,C 180,E1 -19241.373,E2 -19241.373} C_VEL
LIN {X 0,Y 264.407,Z 352.987,A -85,B 0,C 180,E1 -19243.547,E2 -19243.547} C_VEL
LIN {X 0,Y 267.512,Z 358.457,A -85,B 0,C 180,E1 -19245.132,E2 -19245.132} C_VEL
LIN {X 0,Y 271.141,Z 365.412,A -85,B 0,C 180,E1 -19246.827,E2 -19246.827} C_VEL
LIN {X 0,Y 272.44,Z 368.518,A -85,B 0,C 180,E1 -19247.439,E2 -19247.439} C_VEL
LIN {X 0,Y 273.864,Z 383.787,A -85,B 0,C 180,E1 -19248.914,E2 -19248.914} C_VEL
LIN {X 0,Y 273.862,Z 386.129,A -85,B 0,C 180,E1 -19249.073,E2 -19249.073} C_VEL
LIN {X 0,Y 269.001,Z 432.053,A -85,B 0,C 180,E1 -19251.029,E2 -19251.029} C_VEL
LIN {X 0,Y 267.217,Z 444.169,A -85,B 0,C 180,E1 -19251.779,E2 -19251.779} C_VEL
LIN {X 0,Y 265.067,Z 455.278,A -85,B 0,C 180,E1 -19252.766,E2 -19252.766} C_VEL
LIN {X 0,Y 262.808,Z 464.928,A -85,B 0,C 180,E1 -19253.86,E2 -19253.86} C_VEL
LIN {X 0,Y 260.545,Z 473.37,A -85,B 0,C 180,E1 -19255.051,E2 -19255.051} C_VEL
LIN {X 0,Y 258.295,Z 480.679,A -85,B 0,C 180,E1 -19256.296,E2 -19256.296} C_VEL
LIN {X 0,Y 256.087,Z 487.234,A -85,B 0,C 180,E1 -19257.642,E2 -19257.642} C_VEL
LIN {X 0,Y 253.474,Z 494.09,A -85,B 0,C 180,E1 -19259.347,E2 -19259.347} C_VEL
LIN {X 0,Y 250.936,Z 500.149,A -85,B 0,C 180,E1 -19261.204,E2 -19261.204} C_VEL
LIN {X 0,Y 249.447,Z 503.482,A -85,B 0,C 180,E1 -19262.423,E2 -19262.423} C_VEL
LIN {X 0,Y 247.684,Z 507.251,A -85,B 0,C 180,E1 -19264.069,E2 -19264.069} C_VEL
LIN {X 0,Y 245.382,Z 511.521,A -85,B 0,C 180,E1 -19266.579,E2 -19266.579} C_VEL
LIN {X 0,Y 244.076,Z 513.694,A -85,B 0,C 180,E1 -19268.279,E2 -19268.279} C_VEL
LIN {X 0,Y 242.819,Z 515.453,A -85,B 0,C 180,E1 -19270.252,E2 -19270.252} C_VEL
LIN {X 0,Y 241.997,Z 516.212,A -85,B 0,C 180,E1 -19271.73,E2 -19271.73} C_VEL
LIN {X 0,Y 241.221,Z 516.647,A -85,B 0,C 180,E1 -19273.479,E2 -19273.479} C_VEL
LIN {X 0,Y 240.623,Z 516.501,A -85,B 0,C 180,E1 -19275.461,E2 -19275.461} C_VEL
LIN {X 0,Y 240.242,Z 515.967,A -85,B 0,C 180,E1 -19277.011,E2 -19277.011} C_VEL
LIN {X 0,Y 239.951,Z 514.708,A -85,B 0,C 180,E1 -19278.796,E2 -19278.796} C_VEL
LIN {X 0,Y 239.861,Z 511.774,A -85,B 0,C 180,E1 -19281.486,E2 -19281.486} C_VEL
LIN {X 0,Y 240.118,Z 507.247,A -85,B 0,C 180,E1 -19284.191,E2 -19284.191} C_VEL
LIN {X 0,Y 240.388,Z 503.329,A -85,B 0,C 180,E1 -19286.012,E2 -19286.012} C_VEL
LIN {X 0,Y 240.743,Z 498.509,A -85,B 0,C 180,E1 -19287.846,E2 -19287.846} C_VEL
LIN {X 0,Y 241.253,Z 492.646,A -85,B 0,C 180,E1 -19289.686,E2 -19289.686} C_VEL
LIN {X 0,Y 241.9,Z 485.502,A -85,B 0,C 180,E1 -19291.532,E2 -19291.532} C_VEL
LIN {X 0,Y 242.629,Z 477.79,A -85,B 0,C 180,E1 -19293.181,E2 -19293.181} C_VEL
LIN {X 0,Y 243.455,Z 468.812,A -85,B 0,C 180,E1 -19294.761,E2 -19294.761} C_VEL
LIN {X 0,Y 244.442,Z 457.162,A -85,B 0,C 180,E1 -19296.389,E2 -19296.389} C_VEL
LIN {X 0,Y 245.239,Z 446.479,A -85,B 0,C 180,E1 -19297.517,E2 -19297.517} C_VEL
LIN {X 0,Y 245.797,Z 436.109,A -85,B 0,C 180,E1 -19298.357,E2 -19298.357} C_VEL
LIN {X 0,Y 246.366,Z 424.765,A -85,B 0,C 180,E1 -19299.011,E2 -19299.011} C_VEL
LIN {X 0,Y 248.285,Z 372.957,A -85,B 0,C 180,E1 -19301.164,E2 -19301.164} C_VEL
LIN {X 0,Y 244.884,Z 340.469,A -85,B 0,C 180,E1 -19302.765,E2 -19302.765} C_VEL
LIN {X 0,Y 246.058,Z 331.852,A -85,B 0,C 180,E1 -19305.568,E2 -19305.568} C_VEL
LIN {X 0,Y 245.462,Z 327.393,A -85,B 0,C 180,E1 -19307.123,E2 -19307.123} C_VEL
LIN {X 0,Y 243.206,Z 315.955,A -85,B 0,C 180,E1 -19311.283,E2 -19311.283} C_VEL
LIN {X 0,Y 242.036,Z 310.335,A -85,B 0,C 180,E1 -19313.47,E2 -19313.47} C_VEL
LIN {X 0,Y 241.99,Z 310.34,A -85,B 0,C 180,E1 -19317.378,E2 -19317.378} C_VEL
LIN {X 0,Y 241.974,Z 310.342,A -85,B 0,C 180,E1 -19320.616,E2 -19320.616} C_VEL
LIN {X 0,Y 242,Z 310.343,A -85,B 0,C 180,E1 -19324.197,E2 -19324.197} C_VEL
LIN {X 0,Y 241.991,Z 310.343,A -85,B 0,C 180,E1 -19328.337,E2 -19328.337} C_VEL
LIN {X 0,Y 242.12,Z 310.323,A -85,B 0,C 180,E1 -19333.317,E2 -19333.317} C_VEL
LIN {X 0,Y 242.171,Z 310.315,A -85,B 0,C 180,E1 -19338.277,E2 -19338.277} C_VEL
LIN {X 0,Y 242.377,Z 310.292,A -85,B 0,C 180,E1 -19341.661,E2 -19341.661} C_VEL
LIN {X 0,Y 242.401,Z 310.291,A -85,B 0,C 180,E1 -19343.338,E2 -19343.338} C_VEL
LIN {X 0,Y 242.618,Z 310.261,A -85,B 0,C 180,E1 -19348.337,E2 -19348.337} C_VEL
LIN {X 0,Y 242.618,Z 310.264,A -85,B 0,C 180,E1 -19351.656,E2 -19351.656} C_VEL
LIN {X 0,Y 242.402,Z 310.288,A -85,B 0,C 180,E1 -19356.656,E2 -19356.656} C_VEL
LIN {X 0,Y 242.268,Z 310.307,A -85,B 0,C 180,E1 -19360.019,E2 -19360.019} C_VEL
LIN {X 0,Y 242.125,Z 310.323,A -85,B 0,C 180,E1 -19365.138,E2 -19365.138} C_VEL
LIN {X 0,Y 242.028,Z 310.338,A -85,B 0,C 180,E1 -19368.622,E2 -19368.622} C_VEL
LIN {X 0,Y 241.982,Z 310.337,A -85,B 0,C 180,E1 -19372.177,E2 -19372.177} C_VEL
LIN {X 0,Y 242.025,Z 310.335,A -85,B 0,C 180,E1 -19375.815,E2 -19375.815} C_VEL
LIN {X 0,Y 241.958,Z 310.343,A -85,B 0,C 180,E1 -19379.583,E2 -19379.583} C_VEL
LIN {X 0,Y 241.967,Z 310.344,A -85,B 0,C 180,E1 -19383.487,E2 -19383.487} C_VEL
LIN {X 0,Y 241.968,Z 310.343,A -85,B 0,C 180,E1 -19387.577,E2 -19387.577} C_VEL
LIN {X 0,Y 241.911,Z 310.35,A -85,B 0,C 180,E1 -19391.918,E2 -19391.918} C_VEL
LIN {X 0,Y 241.901,Z 310.351,A -85,B 0,C 180,E1 -19396.569,E2 -19396.569} C_VEL
LIN {X 0,Y 241.969,Z 310.341,A -85,B 0,C 180,E1 -19401.636,E2 -19401.636} C_VEL
LIN {X 0,Y 241.952,Z 310.345,A -85,B 0,C 180,E1 -19404.482,E2 -19404.482} C_VEL
LIN {X 0,Y 241.945,Z 310.343,A -85,B 0,C 180,E1 -19408.474,E2 -19408.474} C_VEL
LIN {X 0,Y 241.974,Z 310.341,A -85,B 0,C 180,E1 -19412.307,E2 -19412.307} C_VEL
LIN {X 0,Y 242.004,Z 310.336,A -85,B 0,C 180,E1 -19416.009,E2 -19416.009} C_VEL
LIN {X 0,Y 241.95,Z 310.347,A -85,B 0,C 180,E1 -19419.599,E2 -19419.599} C_VEL
LIN {X 0,Y 242.079,Z 310.328,A -85,B 0,C 180,E1 -19423.315,E2 -19423.315} C_VEL
LIN {X 0,Y 242.128,Z 310.326,A -85,B 0,C 180,E1 -19428.276,E2 -19428.276} C_VEL
LIN {X 0,Y 242.354,Z 310.293,A -85,B 0,C 180,E1 -19431.662,E2 -19431.662} C_VEL
LIN {X 0,Y 242.217,Z 310.311,A -85,B 0,C 180,E1 -19435.005,E2 -19435.005} C_VEL
LIN {X 0,Y 242.597,Z 310.265,A -85,B 0,C 180,E1 -19438.339,E2 -19438.339} C_VEL
LIN {X 0,Y 242.593,Z 310.262,A -85,B 0,C 180,E1 -19441.659,E2 -19441.659} C_VEL
LIN {X 0,Y 242.378,Z 310.291,A -85,B 0,C 180,E1 -19446.659,E2 -19446.659} C_VEL
LIN {X 0,Y 242.228,Z 310.309,A -85,B 0,C 180,E1 -19450.024,E2 -19450.024} C_VEL
LIN {X 0,Y 242.102,Z 310.325,A -85,B 0,C 180,E1 -19455.144,E2 -19455.144} C_VEL
LIN {X 0,Y 242.028,Z 310.333,A -85,B 0,C 180,E1 -19458.627,E2 -19458.627} C_VEL
LIN {X 0,Y 241.969,Z 310.344,A -85,B 0,C 180,E1 -19462.183,E2 -19462.183} C_VEL
LIN {X 0,Y 242.016,Z 310.337,A -85,B 0,C 180,E1 -19465.832,E2 -19465.832} C_VEL
LIN {X 0,Y 241.942,Z 310.342,A -85,B 0,C 180,E1 -19469.591,E2 -19469.591} C_VEL
LIN {X 0,Y 241.937,Z 310.346,A -85,B 0,C 180,E1 -19472.321,E2 -19472.321} C_VEL
LIN {X 0,Y 241.323,Z 310.429,A -85,B 0,C 180,E1 -19473.711,E2 -19473.711} C_VEL
LIN {X 0,Y 238.481,Z 310.785,A -85,B 0,C 180,E1 -19475.976,E2 -19475.976} C_VEL
LIN {X 0,Y 236.015,Z 311.088,A -85,B 0,C 180,E1 -19477.821,E2 -19477.821} C_VEL
LIN {X 0,Y 234.929,Z 311.223,A -85,B 0,C 180,E1 -19479.254,E2 -19479.254} C_VEL
LIN {X 0,Y 234.828,Z 311.231,A -85,B 0,C 180,E1 -19479.741,E2 -19479.741} C_VEL
LIN {X 0,Y 234.856,Z 311.229,A -85,B 0,C 180,E1 -19484.105,E2 -19484.105} C_VEL
LIN {X 0,Y 234.858,Z 311.229,A -85,B 0,C 180,E1 -19488.836,E2 -19488.836} C_VEL
LIN {X 0,Y 234.994,Z 311.391,A -85,B 0,C 180,E1 -19492.937,E2 -19492.937} C_VEL
LIN {X 0,Y 237.438,Z 322.584,A -85,B 0,C 180,E1 -19496.806,E2 -19496.806} C_VEL
LIN {X 0,Y 240.062,Z 334.792,A -85,B 0,C 180,E1 -19500.82,E2 -19500.82} C_VEL
LIN {X 0,Y 240.803,Z 339.038,A -85,B 0,C 180,E1 -19502.169,E2 -19502.169} C_VEL
LIN {X 0,Y 239.939,Z 343.991,A -85,B 0,C 180,E1 -19503.593,E2 -19503.593} C_VEL
LIN {X 0,Y 241.538,Z 368.486,A -85,B 0,C 180,E1 -19504.677,E2 -19504.677} C_VEL
LIN {X 0,Y 242.608,Z 380.591,A -85,B 0,C 180,E1 -19505.219,E2 -19505.219} C_VEL
LIN {X 0,Y 240.355,Z 444.757,A -85,B 0,C 180,E1 -19507.721,E2 -19507.721} C_VEL
LIN {X 0,Y 239.821,Z 454.541,A -85,B 0,C 180,E1 -19508.292,E2 -19508.292} C_VEL
LIN {X 0,Y 239.091,Z 463.773,A -85,B 0,C 180,E1 -19509.013,E2 -19509.013} C_VEL
LIN {X 0,Y 238.262,Z 473.151,A -85,B 0,C 180,E1 -19509.952,E2 -19509.952} C_VEL
LIN {X 0,Y 237.484,Z 481.699,A -85,B 0,C 180,E1 -19511.008,E2 -19511.008} C_VEL
LIN {X 0,Y 236.492,Z 491.287,A -85,B 0,C 180,E1 -19512.466,E2 -19512.466} C_VEL
LIN {X 0,Y 235.583,Z 499.545,A -85,B 0,C 180,E1 -19513.987,E2 -19513.987} C_VEL
LIN {X 0,Y 234.772,Z 507.332,A -85,B 0,C 180,E1 -19515.707,E2 -19515.707} C_VEL
LIN {X 0,Y 234.189,Z 513.947,A -85,B 0,C 180,E1 -19517.438,E2 -19517.438} C_VEL
LIN {X 0,Y 233.644,Z 520.803,A -85,B 0,C 180,E1 -19519.607,E2 -19519.607} C_VEL
LIN {X 0,Y 233.377,Z 525.461,A -85,B 0,C 180,E1 -19521.344,E2 -19521.344} C_VEL
LIN {X 0,Y 233.256,Z 530.875,A -85,B 0,C 180,E1 -19523.866,E2 -19523.866} C_VEL
LIN {X 0,Y 233.212,Z 534.063,A -85,B 0,C 180,E1 -19525.683,E2 -19525.683} C_VEL
LIN {X 0,Y 233.139,Z 537.467,A -85,B 0,C 180,E1 -19528.276,E2 -19528.276} C_VEL
LIN {X 0,Y 233.413,Z 539.057,A -85,B 0,C 180,E1 -19530.003,E2 -19530.003} C_VEL
LIN {X 0,Y 232.956,Z 540.938,A -85,B 0,C 180,E1 -19533.462,E2 -19533.462} C_VEL
LIN {X 0,Y 232.878,Z 540.955,A -85,B 0,C 180,E1 -19536.936,E2 -19536.936} C_VEL
LIN {X 0,Y 233.092,Z 540.448,A -85,B 0,C 180,E1 -19538.673,E2 -19538.673} C_VEL
LIN {X 0,Y 234.08,Z 537.965,A -85,B 0,C 180,E1 -19542.135,E2 -19542.135} C_VEL
LIN {X 0,Y 235.364,Z 535.041,A -85,B 0,C 180,E1 -19544.705,E2 -19544.705} C_VEL
LIN {X 0,Y 237.279,Z 531.065,A -85,B 0,C 180,E1 -19547.231,E2 -19547.231} C_VEL
LIN {X 0,Y 239.46,Z 525.943,A -85,B 0,C 180,E1 -19549.727,E2 -19549.727} C_VEL
LIN {X 0,Y 241.799,Z 520.714,A -85,B 0,C 180,E1 -19551.753,E2 -19551.753} C_VEL
LIN {X 0,Y 244.47,Z 514.484,A -85,B 0,C 180,E1 -19553.734,E2 -19553.734} C_VEL
LIN {X 0,Y 247.517,Z 506.989,A -85,B 0,C 180,E1 -19555.659,E2 -19555.659} C_VEL
LIN {X 0,Y 250.594,Z 498.899,A -85,B 0,C 180,E1 -19557.339,E2 -19557.339} C_VEL
LIN {X 0,Y 253.572,Z 490.305,A -85,B 0,C 180,E1 -19558.788,E2 -19558.788} C_VEL
LIN {X 0,Y 256.281,Z 481.418,A -85,B 0,C 180,E1 -19560.031,E2 -19560.031} C_VEL
LIN {X 0,Y 258.74,Z 472.293,A -85,B 0,C 180,E1 -19561.07,E2 -19561.07} C_VEL
LIN {X 0,Y 260.927,Z 462.985,A -85,B 0,C 180,E1 -19561.911,E2 -19561.911} C_VEL
LIN {X 0,Y 262.941,Z 452.94,A -85,B 0,C 180,E1 -19562.598,E2 -19562.598} C_VEL
LIN {X 0,Y 264.532,Z 442.725,A -85,B 0,C 180,E1 -19563.113,E2 -19563.113} C_VEL
LIN {X 0,Y 269.813,Z 388.313,A -85,B 0,C 180,E1 -19565.212,E2 -19565.212} C_VEL
LIN {X 0,Y 269.262,Z 378.411,A -85,B 0,C 180,E1 -19566.038,E2 -19566.038} C_VEL
LIN {X 0,Y 268.866,Z 376.182,A -85,B 0,C 180,E1 -19566.309,E2 -19566.309} C_VEL
LIN {X 0,Y 265.427,Z 368.313,A -85,B 0,C 180,E1 -19567.983,E2 -19567.983} C_VEL
LIN {X 0,Y 262.273,Z 362.274,A -85,B 0,C 180,E1 -19569.597,E2 -19569.597} C_VEL
LIN {X 0,Y 260.112,Z 358.305,A -85,B 0,C 180,E1 -19570.842,E2 -19570.842} C_VEL
LIN {X 0,Y 257.071,Z 353.178,A -85,B 0,C 180,E1 -19572.744,E2 -19572.744} C_VEL
LIN {X 0,Y 253.487,Z 347.661,A -85,B 0,C 180,E1 -19575.428,E2 -19575.428} C_VEL
LIN {X 0,Y 249.806,Z 342.573,A -85,B 0,C 180,E1 -19579.207,E2 -19579.207} C_VEL
LIN {X 0,Y 248.999,Z 341.053,A -85,B 0,C 180,E1 -19580.672,E2 -19580.672} C_VEL
LIN {X 0,Y 248.668,Z 339.557,A -85,B 0,C 180,E1 -19583.594,E2 -19583.594} C_VEL
LIN {X 0,Y 248.391,Z 339.236,A -85,B 0,C 180,E1 -19588.081,E2 -19588.081} C_VEL
LIN {X 0,Y 248.809,Z 340.019,A -85,B 0,C 180,E1 -19591.303,E2 -19591.303} C_VEL
LIN {X 0,Y 249.337,Z 340.997,A -85,B 0,C 180,E1 -19592.987,E2 -19592.987} C_VEL
LIN {X 0,Y 252.812,Z 345.697,A -85,B 0,C 180,E1 -19596.898,E2 -19596.898} C_VEL
LIN {X 0,Y 254.409,Z 347.928,A -85,B 0,C 180,E1 -19598.264,E2 -19598.264} C_VEL
LIN {X 0,Y 257.986,Z 353.143,A -85,B 0,C 180,E1 -19600.827,E2 -19600.827} C_VEL
LIN {X 0,Y 261.486,Z 358.855,A -85,B 0,C 180,E1 -19602.952,E2 -19602.952} C_VEL
LIN {X 0,Y 264.692,Z 364.759,A -85,B 0,C 180,E1 -19604.682,E2 -19604.682} C_VEL
LIN {X 0,Y 268.109,Z 371.974,A -85,B 0,C 180,E1 -19606.415,E2 -19606.415} C_VEL
LIN {X 0,Y 269.074,Z 381.041,A -85,B 0,C 180,E1 -19607.394,E2 -19607.394} C_VEL
LIN {X 0,Y 269.362,Z 387.033,A -85,B 0,C 180,E1 -19607.926,E2 -19607.926} C_VEL
LIN {X 0,Y 264.191,Z 433.035,A -85,B 0,C 180,E1 -19609.931,E2 -19609.931} C_VEL
LIN {X 0,Y 262.186,Z 445.729,A -85,B 0,C 180,E1 -19610.746,E2 -19610.746} C_VEL
LIN {X 0,Y 259.726,Z 457.399,A -85,B 0,C 180,E1 -19611.834,E2 -19611.834} C_VEL
LIN {X 0,Y 257.709,Z 465.32,A -85,B 0,C 180,E1 -19612.755,E2 -19612.755} C_VEL
LIN {X 0,Y 255.363,Z 473.481,A -85,B 0,C 180,E1 -19613.924,E2 -19613.924} C_VEL
LIN {X 0,Y 252.551,Z 481.969,A -85,B 0,C 180,E1 -19615.412,E2 -19615.412} C_VEL
LIN {X 0,Y 250.21,Z 488.419,A -85,B 0,C 180,E1 -19616.78,E2 -19616.78} C_VEL
LIN {X 0,Y 247.672,Z 494.671,A -85,B 0,C 180,E1 -19618.375,E2 -19618.375} C_VEL
LIN {X 0,Y 245.326,Z 499.919,A -85,B 0,C 180,E1 -19620.001,E2 -19620.001} C_VEL
LIN {X 0,Y 243.172,Z 504.327,A -85,B 0,C 180,E1 -19621.657,E2 -19621.657} C_VEL
LIN {X 0,Y 240.496,Z 509.337,A -85,B 0,C 180,E1 -19624.084,E2 -19624.084} C_VEL
LIN {X 0,Y 238.815,Z 512.202,A -85,B 0,C 180,E1 -19625.913,E2 -19625.913} C_VEL
LIN {X 0,Y 236.756,Z 515.099,A -85,B 0,C 180,E1 -19628.536,E2 -19628.536} C_VEL
LIN {X 0,Y 235.671,Z 516.316,A -85,B 0,C 180,E1 -19630.308,E2 -19630.308} C_VEL
LIN {X 0,Y 234.723,Z 517.044,A -85,B 0,C 180,E1 -19632.099,E2 -19632.099} C_VEL
LIN {X 0,Y 233.99,Z 517.19,A -85,B 0,C 180,E1 -19633.904,E2 -19633.904} C_VEL
LIN {X 0,Y 233.454,Z 516.712,A -85,B 0,C 180,E1 -19635.721,E2 -19635.721} C_VEL
LIN {X 0,Y 233.025,Z 515.716,A -85,B 0,C 180,E1 -19637.555,E2 -19637.555} C_VEL
LIN {X 0,Y 232.79,Z 512.822,A -85,B 0,C 180,E1 -19640.632,E2 -19640.632} C_VEL
LIN {X 0,Y 232.873,Z 509.25,A -85,B 0,C 180,E1 -19643.101,E2 -19643.101} C_VEL
LIN {X 0,Y 233.187,Z 505.017,A -85,B 0,C 180,E1 -19645.293,E2 -19645.293} C_VEL
LIN {X 0,Y 233.644,Z 498.722,A -85,B 0,C 180,E1 -19647.791,E2 -19647.791} C_VEL
LIN {X 0,Y 234.21,Z 492.027,A -85,B 0,C 180,E1 -19649.909,E2 -19649.909} C_VEL
LIN {X 0,Y 234.907,Z 484.62,A -85,B 0,C 180,E1 -19651.825,E2 -19651.825} C_VEL
LIN {X 0,Y 235.623,Z 476.845,A -85,B 0,C 180,E1 -19653.487,E2 -19653.487} C_VEL
LIN {X 0,Y 236.669,Z 465.847,A -85,B 0,C 180,E1 -19655.386,E2 -19655.386} C_VEL
LIN {X 0,Y 237.432,Z 456.316,A -85,B 0,C 180,E1 -19656.669,E2 -19656.669} C_VEL
LIN {X 0,Y 238.164,Z 447.132,A -85,B 0,C 180,E1 -19657.663,E2 -19657.663} C_VEL
LIN {X 0,Y 238.786,Z 436.616,A -85,B 0,C 180,E1 -19658.547,E2 -19658.547} C_VEL
LIN {X 0,Y 239.324,Z 425.482,A -85,B 0,C 180,E1 -19659.22,E2 -19659.22} C_VEL
LIN {X 0,Y 241.281,Z 373.338,A -85,B 0,C 180,E1 -19661.487,E2 -19661.487} C_VEL
LIN {X 0,Y 237.928,Z 340.664,A -85,B 0,C 180,E1 -19663.123,E2 -19663.123} C_VEL
LIN {X 0,Y 239.051,Z 332.286,A -85,B 0,C 180,E1 -19665.908,E2 -19665.908} C_VEL
LIN {X 0,Y 237.321,Z 322.87,A -85,B 0,C 180,E1 -19669.345,E2 -19669.345} C_VEL
LIN {X 0,Y 235.231,Z 312.507,A -85,B 0,C 180,E1 -19673.306,E2 -19673.306} C_VEL
LIN {X 0,Y 234.988,Z 311.213,A -85,B 0,C 180,E1 -19673.855,E2 -19673.855} C_VEL
LIN {X 0,Y 234.955,Z 311.217,A -85,B 0,C 180,E1 -19677.424,E2 -19677.424} C_VEL
LIN {X 0,Y 234.894,Z 311.224,A -85,B 0,C 180,E1 -19681.398,E2 -19681.398} C_VEL
LIN {X 0,Y 234.918,Z 311.221,A -85,B 0,C 180,E1 -19685.238,E2 -19685.238} C_VEL
LIN {X 0,Y 234.945,Z 311.218,A -85,B 0,C 180,E1 -19688.962,E2 -19688.962} C_VEL
LIN {X 0,Y 235.061,Z 311.204,A -85,B 0,C 180,E1 -19693.092,E2 -19693.092} C_VEL
LIN {X 0,Y 235.103,Z 311.196,A -85,B 0,C 180,E1 -19697.919,E2 -19697.919} C_VEL
LIN {X 0,Y 235.317,Z 311.173,A -85,B 0,C 180,E1 -19701.409,E2 -19701.409} C_VEL
LIN {X 0,Y 235.352,Z 311.168,A -85,B 0,C 180,E1 -19703.137,E2 -19703.137} C_VEL
LIN {X 0,Y 235.577,Z 311.138,A -85,B 0,C 180,E1 -19708.287,E2 -19708.287} C_VEL
LIN {X 0,Y 235.577,Z 311.141,A -85,B 0,C 180,E1 -19711.706,E2 -19711.706} C_VEL
LIN {X 0,Y 235.354,Z 311.166,A -85,B 0,C 180,E1 -19716.856,E2 -19716.856} C_VEL
LIN {X 0,Y 235.215,Z 311.186,A -85,B 0,C 180,E1 -19720.323,E2 -19720.323} C_VEL
LIN {X 0,Y 235.073,Z 311.2,A -85,B 0,C 180,E1 -19725.604,E2 -19725.604} C_VEL
LIN {X 0,Y 234.966,Z 311.215,A -85,B 0,C 180,E1 -19729.203,E2 -19729.203} C_VEL
LIN {X 0,Y 234.932,Z 311.219,A -85,B 0,C 180,E1 -19732.88,E2 -19732.88} C_VEL
LIN {X 0,Y 234.937,Z 311.218,A -85,B 0,C 180,E1 -19736.655,E2 -19736.655} C_VEL
LIN {X 0,Y 234.888,Z 311.22,A -85,B 0,C 180,E1 -19740.567,E2 -19740.567} C_VEL
LIN {X 0,Y 234.912,Z 311.221,A -85,B 0,C 180,E1 -19744.633,E2 -19744.633} C_VEL
LIN {X 0,Y 234.896,Z 311.22,A -85,B 0,C 180,E1 -19748.929,E2 -19748.929} C_VEL
LIN {X 0,Y 234.858,Z 311.228,A -85,B 0,C 180,E1 -19753.482,E2 -19753.482} C_VEL
LIN {X 0,Y 234.854,Z 311.23,A -85,B 0,C 180,E1 -19756.505,E2 -19756.505} C_VEL
LIN {X 0,Y 234.895,Z 311.224,A -85,B 0,C 180,E1 -19761.073,E2 -19761.073} C_VEL
LIN {X 0,Y 234.898,Z 311.222,A -85,B 0,C 180,E1 -19765.355,E2 -19765.355} C_VEL
LIN {X 0,Y 234.902,Z 311.224,A -85,B 0,C 180,E1 -19769.427,E2 -19769.427} C_VEL
LIN {X 0,Y 234.964,Z 311.215,A -85,B 0,C 180,E1 -19773.79,E2 -19773.79} C_VEL
LIN {X 0,Y 234.92,Z 311.221,A -85,B 0,C 180,E1 -19778.011,E2 -19778.011} C_VEL
LIN {X 0,Y 235.02,Z 311.206,A -85,B 0,C 180,E1 -19783.091,E2 -19783.091} C_VEL
LIN {X 0,Y 235.06,Z 311.204,A -85,B 0,C 180,E1 -19787.918,E2 -19787.918} C_VEL
LIN {X 0,Y 235.282,Z 311.174,A -85,B 0,C 180,E1 -19791.41,E2 -19791.41} C_VEL
LIN {X 0,Y 235.329,Z 311.166,A -85,B 0,C 180,E1 -19793.138,E2 -19793.138} C_VEL
LIN {X 0,Y 235.557,Z 311.141,A -85,B 0,C 180,E1 -19798.289,E2 -19798.289} C_VEL
LIN {X 0,Y 235.552,Z 311.139,A -85,B 0,C 180,E1 -19801.709,E2 -19801.709} C_VEL
LIN {X 0,Y 235.329,Z 311.17,A -85,B 0,C 180,E1 -19806.86,E2 -19806.86} C_VEL
LIN {X 0,Y 235.174,Z 311.186,A -85,B 0,C 180,E1 -19810.328,E2 -19810.328} C_VEL
LIN {X 0,Y 235.056,Z 311.206,A -85,B 0,C 180,E1 -19815.609,E2 -19815.609} C_VEL
LIN {X 0,Y 234.966,Z 311.213,A -85,B 0,C 180,E1 -19819.208,E2 -19819.208} C_VEL
LIN {X 0,Y 234.916,Z 311.22,A -85,B 0,C 180,E1 -19822.886,E2 -19822.886} C_VEL
LIN {X 0,Y 234.922,Z 311.221,A -85,B 0,C 180,E1 -19826.662,E2 -19826.662} C_VEL
LIN {X 0,Y 234.869,Z 311.227,A -85,B 0,C 180,E1 -19830.576,E2 -19830.576} C_VEL
LIN {X 0,Y 234.894,Z 311.226,A -85,B 0,C 180,E1 -19834.643,E2 -19834.643} C_VEL
LIN {X 0,Y 234.884,Z 311.228,A -85,B 0,C 180,E1 -19838.939,E2 -19838.939} C_VEL
LIN {X 0,Y 234.828,Z 311.231,A -85,B 0,C 180,E1 -19839.741,E2 -19839.741} C_VEL
LIN {X 0,Y 234.129,Z 311.323,A -85,B 0,C 180,E1 -19841.173,E2 -19841.173} C_VEL
LIN {X 0,Y 231.281,Z 311.677,A -85,B 0,C 180,E1 -19843.51,E2 -19843.51} C_VEL
LIN {X 0,Y 228.884,Z 311.976,A -85,B 0,C 180,E1 -19845.415,E2 -19845.415} C_VEL
LIN {X 0,Y 227.862,Z 312.102,A -85,B 0,C 180,E1 -19846.893,E2 -19846.893} C_VEL
LIN {X 0,Y 227.78,Z 312.112,A -85,B 0,C 180,E1 -19847.394,E2 -19847.394} C_VEL
LIN {X 0,Y 227.942,Z 312.254,A -85,B 0,C 180,E1 -19852.469,E2 -19852.469} C_VEL
LIN {X 0,Y 230.549,Z 324.21,A -85,B 0,C 180,E1 -19856.73,E2 -19856.73} C_VEL
LIN {X 0,Y 233.187,Z 336.596,A -85,B 0,C 180,E1 -19860.928,E2 -19860.928} C_VEL
LIN {X 0,Y 233.701,Z 340.613,A -85,B 0,C 180,E1 -19862.224,E2 -19862.224} C_VEL
LIN {X 0,Y 233.04,Z 343.855,A -85,B 0,C 180,E1 -19863.2,E2 -19863.2} C_VEL
LIN {X 0,Y 234.339,Z 365.701,A -85,B 0,C 180,E1 -19864.2,E2 -19864.2} C_VEL
LIN {X 0,Y 235.621,Z 381.704,A -85,B 0,C 180,E1 -19864.934,E2 -19864.934} C_VEL
LIN {X 0,Y 233.326,Z 444.734,A -85,B 0,C 180,E1 -19867.48,E2 -19867.48} C_VEL
LIN {X 0,Y 232.736,Z 455.172,A -85,B 0,C 180,E1 -19868.121,E2 -19868.121} C_VEL
LIN {X 0,Y 231.957,Z 464.747,A -85,B 0,C 180,E1 -19868.918,E2 -19868.918} C_VEL
LIN {X 0,Y 231.212,Z 472.951,A -85,B 0,C 180,E1 -19869.778,E2 -19869.778} C_VEL
LIN {X 0,Y 230.358,Z 482.046,A -85,B 0,C 180,E1 -19870.949,E2 -19870.949} C_VEL
LIN {X 0,Y 229.389,Z 491.197,A -85,B 0,C 180,E1 -19872.395,E2 -19872.395} C_VEL
LIN {X 0,Y 228.509,Z 499.288,A -85,B 0,C 180,E1 -19873.936,E2 -19873.936} C_VEL
LIN {X 0,Y 227.672,Z 507.055,A -85,B 0,C 180,E1 -19875.708,E2 -19875.708} C_VEL
LIN {X 0,Y 227.094,Z 513.656,A -85,B 0,C 180,E1 -19877.494,E2 -19877.494} C_VEL
LIN {X 0,Y 226.569,Z 520.49,A -85,B 0,C 180,E1 -19879.73,E2 -19879.73} C_VEL
LIN {X 0,Y 226.282,Z 526.09,A -85,B 0,C 180,E1 -19881.97,E2 -19881.97} C_VEL
LIN {X 0,Y 226.225,Z 531.415,A -85,B 0,C 180,E1 -19884.656,E2 -19884.656} C_VEL
LIN {X 0,Y 226.096,Z 535.393,A -85,B 0,C 180,E1 -19887.331,E2 -19887.331} C_VEL
LIN {X 0,Y 226.358,Z 538.23,A -85,B 0,C 180,E1 -19890.004,E2 -19890.004} C_VEL
LIN {X 0,Y 225.91,Z 539.486,A -85,B 0,C 180,E1 -19891.786,E2 -19891.786} C_VEL
LIN {X 0,Y 225.888,Z 540.315,A -85,B 0,C 180,E1 -19893.571,E2 -19893.571} C_VEL
LIN {X 0,Y 225.806,Z 540.599,A -85,B 0,C 180,E1 -19897.155,E2 -19897.155} C_VEL
LIN {X 0,Y 226.059,Z 540.107,A -85,B 0,C 180,E1 -19898.945,E2 -19898.945} C_VEL
LIN {X 0,Y 227.096,Z 537.952,A -85,B 0,C 180,E1 -19902.514,E2 -19902.514} C_VEL
LIN {X 0,Y 228.493,Z 535.197,A -85,B 0,C 180,E1 -19905.158,E2 -19905.158} C_VEL
LIN {X 0,Y 230.522,Z 531.395,A -85,B 0,C 180,E1 -19907.752,E2 -19907.752} C_VEL
LIN {X 0,Y 233.195,Z 525.653,A -85,B 0,C 180,E1 -19910.694,E2 -19910.694} C_VEL
LIN {X 0,Y 235.769,Z 520.376,A -85,B 0,C 180,E1 -19912.801,E2 -19912.801} C_VEL
LIN {X 0,Y 238.717,Z 514.139,A -85,B 0,C 180,E1 -19914.806,E2 -19914.806} C_VEL
LIN {X 0,Y 241.901,Z 506.656,A -85,B 0,C 180,E1 -19916.765,E2 -19916.765} C_VEL
LIN {X 0,Y 244.83,Z 499.654,A -85,B 0,C 180,E1 -19918.272,E2 -19918.272} C_VEL
LIN {X 0,Y 247.938,Z 491.383,A -85,B 0,C 180,E1 -19919.74,E2 -19919.74} C_VEL
LIN {X 0,Y 250.774,Z 482.812,A -85,B 0,C 180,E1 -19920.995,E2 -19920.995} C_VEL
LIN {X 0,Y 253.771,Z 472.348,A -85,B 0,C 180,E1 -19922.216,E2 -19922.216} C_VEL
LIN {X 0,Y 256.073,Z 463.122,A -85,B 0,C 180,E1 -19923.057,E2 -19923.057} C_VEL
LIN {X 0,Y 258.419,Z 451.928,A -85,B 0,C 180,E1 -19923.826,E2 -19923.826} C_VEL
LIN {X 0,Y 260.073,Z 441.698,A -85,B 0,C 180,E1 -19924.34,E2 -19924.34} C_VEL
LIN {X 0,Y 265.478,Z 389.551,A -85,B 0,C 180,E1 -19926.391,E2 -19926.391} C_VEL
LIN {X 0,Y 265.018,Z 380.622,A -85,B 0,C 180,E1 -19927.171,E2 -19927.171} C_VEL
LIN {X 0,Y 261.882,Z 373.12,A -85,B 0,C 180,E1 -19928.847,E2 -19928.847} C_VEL
LIN {X 0,Y 259.376,Z 368.016,A -85,B 0,C 180,E1 -19930.254,E2 -19930.254} C_VEL
LIN {X 0,Y 257.069,Z 363.657,A -85,B 0,C 180,E1 -19931.663,E2 -19931.663} C_VEL
LIN {X 0,Y 254.638,Z 359.375,A -85,B 0,C 180,E1 -19933.323,E2 -19933.323} C_VEL
LIN {X 0,Y 251.284,Z 353.9,A -85,B 0,C 180,E1 -19936.046,E2 -19936.046} C_VEL
LIN {X 0,Y 247.816,Z 348.819,A -85,B 0,C 180,E1 -19939.969,E2 -19939.969} C_VEL
LIN {X 0,Y 246.733,Z 347.161,A -85,B 0,C 180,E1 -19941.909,E2 -19941.909} C_VEL
LIN {X 0,Y 245.92,Z 346.06,A -85,B 0,C 180,E1 -19944.137,E2 -19944.137} C_VEL
LIN {X 0,Y 245.624,Z 345.791,A -85,B 0,C 180,E1 -19947.069,E2 -19947.069} C_VEL
LIN {X 0,Y 246.29,Z 346.345,A -85,B 0,C 180,E1 -19950.043,E2 -19950.043} C_VEL
LIN {X 0,Y 247.658,Z 347.778,A -85,B 0,C 180,E1 -19952.685,E2 -19952.685} C_VEL
LIN {X 0,Y 251.208,Z 352.729,A -85,B 0,C 180,E1 -19956.842,E2 -19956.842} C_VEL
LIN {X 0,Y 255.46,Z 359.267,A -85,B 0,C 180,E1 -19960.266,E2 -19960.266} C_VEL
LIN {X 0,Y 258.742,Z 364.935,A -85,B 0,C 180,E1 -19962.393,E2 -19962.393} C_VEL
LIN {X 0,Y 261.579,Z 370.487,A -85,B 0,C 180,E1 -19964.063,E2 -19964.063} C_VEL
LIN {X 0,Y 264.282,Z 376.471,A -85,B 0,C 180,E1 -19965.543,E2 -19965.543} C_VEL
LIN {X 0,Y 265.036,Z 388.045,A -85,B 0,C 180,E1 -19966.729,E2 -19966.729} C_VEL
LIN {X 0,Y 259.743,Z 432.936,A -85,B 0,C 180,E1 -19968.711,E2 -19968.711} C_VEL
LIN {X 0,Y 257.784,Z 444.775,A -85,B 0,C 180,E1 -19969.46,E2 -19969.46} C_VEL
LIN {X 0,Y 255.28,Z 456.203,A -85,B 0,C 180,E1 -19970.493,E2 -19970.493} C_VEL
LIN {X 0,Y 252.737,Z 465.782,A -85,B 0,C 180,E1 -19971.606,E2 -19971.606} C_VEL
LIN {X 0,Y 249.948,Z 474.888,A -85,B 0,C 180,E1 -19972.935,E2 -19972.935} C_VEL
LIN {X 0,Y 247.168,Z 482.782,A -85,B 0,C 180,E1 -19974.356,E2 -19974.356} C_VEL
LIN {X 0,Y 243.713,Z 491.402,A -85,B 0,C 180,E1 -19976.281,E2 -19976.281} C_VEL
LIN {X 0,Y 239.94,Z 499.547,A -85,B 0,C 180,E1 -19978.68,E2 -19978.68} C_VEL
LIN {X 0,Y 238.003,Z 503.405,A -85,B 0,C 180,E1 -19980.06,E2 -19980.06} C_VEL
LIN {X 0,Y 234.898,Z 508.831,A -85,B 0,C 180,E1 -19982.573,E2 -19982.573} C_VEL
LIN {X 0,Y 232.285,Z 512.906,A -85,B 0,C 180,E1 -19985.209,E2 -19985.209} C_VEL
LIN {X 0,Y 230.765,Z 514.932,A -85,B 0,C 180,E1 -19986.998,E2 -19986.998} C_VEL
LIN {X 0,Y 229.453,Z 516.438,A -85,B 0,C 180,E1 -19988.81,E2 -19988.81} C_VEL
LIN {X 0,Y 228.348,Z 517.297,A -85,B 0,C 180,E1 -19990.643,E2 -19990.643} C_VEL
LIN {X 0,Y 227.421,Z 517.605,A -85,B 0,C 180,E1 -19992.494,E2 -19992.494} C_VEL
LIN {X 0,Y 226.341,Z 516.991,A -85,B 0,C 180,E1 -19995.734,E2 -19995.734} C_VEL
LIN {X 0,Y 225.845,Z 515.429,A -85,B 0,C 180,E1 -19998.132,E2 -19998.132} C_VEL
LIN {X 0,Y 225.696,Z 512.432,A -85,B 0,C 180,E1 -20000.909,E2 -20000.909} C_VEL
LIN {X 0,Y 225.765,Z 509.484,A -85,B 0,C 180,E1 -20002.901,E2 -20002.901} C_VEL
LIN {X 0,Y 226.167,Z 503.949,A -85,B 0,C 180,E1 -20005.693,E2 -20005.693} C_VEL
LIN {X 0,Y 226.538,Z 498.844,A -85,B 0,C 180,E1 -20007.734,E2 -20007.734} C_VEL
LIN {X 0,Y 227.127,Z 491.986,A -85,B 0,C 180,E1 -20009.959,E2 -20009.959} C_VEL
LIN {X 0,Y 227.709,Z 485.704,A -85,B 0,C 180,E1 -20011.648,E2 -20011.648} C_VEL
LIN {X 0,Y 228.451,Z 478.082,A -85,B 0,C 180,E1 -20013.361,E2 -20013.361} C_VEL
LIN {X 0,Y 229.35,Z 468.813,A -85,B 0,C 180,E1 -20015.072,E2 -20015.072} C_VEL
LIN {X 0,Y 230.343,Z 456.993,A -85,B 0,C 180,E1 -20016.784,E2 -20016.784} C_VEL
LIN {X 0,Y 231.173,Z 446.598,A -85,B 0,C 180,E1 -20017.933,E2 -20017.933} C_VEL
LIN {X 0,Y 231.758,Z 436.403,A -85,B 0,C 180,E1 -20018.803,E2 -20018.803} C_VEL
LIN {X 0,Y 232.405,Z 423.836,A -85,B 0,C 180,E1 -20019.565,E2 -20019.565} C_VEL
LIN {X 0,Y 234.297,Z 373.857,A -85,B 0,C 180,E1 -20021.794,E2 -20021.794} C_VEL
LIN {X 0,Y 230.99,Z 340.647,A -85,B 0,C 180,E1 -20023.53,E2 -20023.53} C_VEL
LIN {X 0,Y 232.006,Z 333.895,A -85,B 0,C 180,E1 -20025.836,E2 -20025.836} C_VEL
LIN {X 0,Y 231.462,Z 329.772,A -85,B 0,C 180,E1 -20027.352,E2 -20027.352} C_VEL
LIN {X 0,Y 229.27,Z 318.582,A -85,B 0,C 180,E1 -20031.63,E2 -20031.63} C_VEL
LIN {X 0,Y 227.917,Z 312.092,A -85,B 0,C 180,E1 -20034.271,E2 -20034.271} C_VEL
LIN {X 0,Y 227.857,Z 312.101,A -85,B 0,C 180,E1 -20038.375,E2 -20038.375} C_VEL
LIN {X 0,Y 227.837,Z 312.105,A -85,B 0,C 180,E1 -20042.438,E2 -20042.438} C_VEL
LIN {X 0,Y 227.87,Z 312.103,A -85,B 0,C 180,E1 -20046.361,E2 -20046.361} C_VEL
LIN {X 0,Y 227.901,Z 312.096,A -85,B 0,C 180,E1 -20050.169,E2 -20050.169} C_VEL
LIN {X 0,Y 228.024,Z 312.078,A -85,B 0,C 180,E1 -20053.893,E2 -20053.893} C_VEL
LIN {X 0,Y 228.148,Z 312.066,A -85,B 0,C 180,E1 -20059.346,E2 -20059.346} C_VEL
LIN {X 0,Y 228.305,Z 312.045,A -85,B 0,C 180,E1 -20062.924,E2 -20062.924} C_VEL
LIN {X 0,Y 228.535,Z 312.016,A -85,B 0,C 180,E1 -20068.234,E2 -20068.234} C_VEL
LIN {X 0,Y 228.535,Z 312.018,A -85,B 0,C 180,E1 -20071.759,E2 -20071.759} C_VEL
LIN {X 0,Y 228.307,Z 312.043,A -85,B 0,C 180,E1 -20077.069,E2 -20077.069} C_VEL
LIN {X 0,Y 228.146,Z 312.064,A -85,B 0,C 180,E1 -20080.646,E2 -20080.646} C_VEL
LIN {X 0,Y 228.04,Z 312.076,A -85,B 0,C 180,E1 -20084.268,E2 -20084.268} C_VEL
LIN {X 0,Y 227.927,Z 312.091,A -85,B 0,C 180,E1 -20087.954,E2 -20087.954} C_VEL
LIN {X 0,Y 227.898,Z 312.091,A -85,B 0,C 180,E1 -20092.307,E2 -20092.307} C_VEL
LIN {X 0,Y 227.915,Z 312.093,A -85,B 0,C 180,E1 -20096.586,E2 -20096.586} C_VEL
LIN {X 0,Y 227.863,Z 312.095,A -85,B 0,C 180,E1 -20100.274,E2 -20100.274} C_VEL
LIN {X 0,Y 227.864,Z 312.103,A -85,B 0,C 180,E1 -20103.714,E2 -20103.714} C_VEL
LIN {X 0,Y 227.825,Z 312.104,A -85,B 0,C 180,E1 -20108.086,E2 -20108.086} C_VEL
LIN {X 0,Y 227.785,Z 312.109,A -85,B 0,C 180,E1 -20112.738,E2 -20112.738} C_VEL
LIN {X 0,Y 227.78,Z 312.107,A -85,B 0,C 180,E1 -20117.249,E2 -20117.249} C_VEL
LIN {X 0,Y 227.816,Z 312.105,A -85,B 0,C 180,E1 -20121.902,E2 -20121.902} C_VEL
LIN {X 0,Y 227.853,Z 312.099,A -85,B 0,C 180,E1 -20126.372,E2 -20126.372} C_VEL
LIN {X 0,Y 227.89,Z 312.095,A -85,B 0,C 180,E1 -20130.433,E2 -20130.433} C_VEL
LIN {X 0,Y 227.894,Z 312.094,A -85,B 0,C 180,E1 -20134.421,E2 -20134.421} C_VEL
LIN {X 0,Y 227.884,Z 312.096,A -85,B 0,C 180,E1 -20138.278,E2 -20138.278} C_VEL
LIN {X 0,Y 227.982,Z 312.086,A -85,B 0,C 180,E1 -20143.891,E2 -20143.891} C_VEL
LIN {X 0,Y 228.105,Z 312.069,A -85,B 0,C 180,E1 -20149.346,E2 -20149.346} C_VEL
LIN {X 0,Y 228.279,Z 312.045,A -85,B 0,C 180,E1 -20152.925,E2 -20152.925} C_VEL
LIN {X 0,Y 228.516,Z 312.018,A -85,B 0,C 180,E1 -20158.237,E2 -20158.237} C_VEL
LIN {X 0,Y 228.512,Z 312.016,A -85,B 0,C 180,E1 -20161.761,E2 -20161.761} C_VEL
LIN {X 0,Y 228.28,Z 312.05,A -85,B 0,C 180,E1 -20167.073,E2 -20167.073} C_VEL
LIN {X 0,Y 228.105,Z 312.067,A -85,B 0,C 180,E1 -20170.652,E2 -20170.652} C_VEL
LIN {X 0,Y 228.007,Z 312.083,A -85,B 0,C 180,E1 -20176.105,E2 -20176.105} C_VEL
LIN {X 0,Y 227.897,Z 312.096,A -85,B 0,C 180,E1 -20179.829,E2 -20179.829} C_VEL
LIN {X 0,Y 227.868,Z 312.098,A -85,B 0,C 180,E1 -20183.637,E2 -20183.637} C_VEL
LIN {X 0,Y 227.832,Z 312.102,A -85,B 0,C 180,E1 -20187.561,E2 -20187.561} C_VEL
LIN {X 0,Y 227.825,Z 312.103,A -85,B 0,C 180,E1 -20191.628,E2 -20191.628} C_VEL
LIN {X 0,Y 227.835,Z 312.101,A -85,B 0,C 180,E1 -20195.879,E2 -20195.879} C_VEL
LIN {X 0,Y 227.782,Z 312.11,A -85,B 0,C 180,E1 -20200.385,E2 -20200.385} C_VEL
LIN {X 0,Y 227.8,Z 312.11,A -85,B 0,C 180,E1 -20205.2,E2 -20205.2} C_VEL
LIN {X 0,Y 227.78,Z 312.112,A -85,B 0,C 180,E1 -20207.394,E2 -20207.394} C_VEL
LIN {X 0,Y 227.07,Z 312.232,A -85,B 0,C 180,E1 -20208.421,E2 -20208.421} C_VEL
LIN {X 0,Y 221.534,Z 313.061,A -85,B 0,C 180,E1 -20211.619,E2 -20211.619} C_VEL
LIN {X 0,Y 221.126,Z 314.166,A -85,B 0,C 180,E1 -20212.388,E2 -20212.388} C_VEL
LIN {X 0,Y 221.174,Z 314.505,A -85,B 0,C 180,E1 -20212.528,E2 -20212.528} C_VEL
LIN {X 0,Y 223.632,Z 325.764,A -85,B 0,C 180,E1 -20216.645,E2 -20216.645} C_VEL
LIN {X 0,Y 226.187,Z 337.647,A -85,B 0,C 180,E1 -20220.785,E2 -20220.785} C_VEL
LIN {X 0,Y 226.665,Z 340.62,A -85,B 0,C 180,E1 -20221.788,E2 -20221.788} C_VEL
LIN {X 0,Y 226.169,Z 343.731,A -85,B 0,C 180,E1 -20222.767,E2 -20222.767} C_VEL
LIN {X 0,Y 227.307,Z 365.04,A -85,B 0,C 180,E1 -20223.789,E2 -20223.789} C_VEL
LIN {X 0,Y 228.677,Z 381.614,A -85,B 0,C 180,E1 -20224.583,E2 -20224.583} C_VEL
LIN {X 0,Y 226.377,Z 443.609,A -85,B 0,C 180,E1 -20227.172,E2 -20227.172} C_VEL
LIN {X 0,Y 225.821,Z 453.478,A -85,B 0,C 180,E1 -20227.776,E2 -20227.776} C_VEL
LIN {X 0,Y 225.023,Z 463.328,A -85,B 0,C 180,E1 -20228.597,E2 -20228.597} C_VEL
LIN {X 0,Y 224.162,Z 472.617,A -85,B 0,C 180,E1 -20229.592,E2 -20229.592} C_VEL
LIN {X 0,Y 223.285,Z 481.919,A -85,B 0,C 180,E1 -20230.837,E2 -20230.837} C_VEL
LIN {X 0,Y 222.326,Z 490.812,A -85,B 0,C 180,E1 -20232.292,E2 -20232.292} C_VEL
LIN {X 0,Y 221.448,Z 498.889,A -85,B 0,C 180,E1 -20233.883,E2 -20233.883} C_VEL
LIN {X 0,Y 220.584,Z 506.632,A -85,B 0,C 180,E1 -20235.71,E2 -20235.71} C_VEL
LIN {X 0,Y 220.026,Z 513.229,A -85,B 0,C 180,E1 -20237.554,E2 -20237.554} C_VEL
LIN {X 0,Y 219.504,Z 520.059,A -85,B 0,C 180,E1 -20239.862,E2 -20239.862} C_VEL
LIN {X 0,Y 219.268,Z 524.694,A -85,B 0,C 180,E1 -20241.712,E2 -20241.712} C_VEL
LIN {X 0,Y 219.173,Z 530.223,A -85,B 0,C 180,E1 -20244.484,E2 -20244.484} C_VEL
LIN {X 0,Y 219.061,Z 533.222,A -85,B 0,C 180,E1 -20246.325,E2 -20246.325} C_VEL
LIN {X 0,Y 219.061,Z 535.522,A -85,B 0,C 180,E1 -20248.165,E2 -20248.165} C_VEL
LIN {X 0,Y 219.303,Z 537.404,A -85,B 0,C 180,E1 -20250.004,E2 -20250.004} C_VEL
LIN {X 0,Y 218.842,Z 538.81,A -85,B 0,C 180,E1 -20251.844,E2 -20251.844} C_VEL
LIN {X 0,Y 218.688,Z 540.043,A -85,B 0,C 180,E1 -20254.975,E2 -20254.975} C_VEL
LIN {X 0,Y 218.759,Z 540.212,A -85,B 0,C 180,E1 -20257.386,E2 -20257.386} C_VEL
LIN {X 0,Y 219.475,Z 538.998,A -85,B 0,C 180,E1 -20261.08,E2 -20261.08} C_VEL
LIN {X 0,Y 220.124,Z 537.856,A -85,B 0,C 180,E1 -20262.917,E2 -20262.917} C_VEL
LIN {X 0,Y 222.277,Z 534.167,A -85,B 0,C 180,E1 -20266.535,E2 -20266.535} C_VEL
LIN {X 0,Y 224.555,Z 530.247,A -85,B 0,C 180,E1 -20269.187,E2 -20269.187} C_VEL
LIN {X 0,Y 227.212,Z 525.006,A -85,B 0,C 180,E1 -20271.886,E2 -20271.886} C_VEL
LIN {X 0,Y 230.449,Z 518.865,A -85,B 0,C 180,E1 -20274.313,E2 -20274.313} C_VEL
LIN {X 0,Y 233.066,Z 513.885,A -85,B 0,C 180,E1 -20275.929,E2 -20275.929} C_VEL
LIN {X 0,Y 236.433,Z 506.527,A -85,B 0,C 180,E1 -20277.916,E2 -20277.916} C_VEL
LIN {X 0,Y 239.521,Z 499.56,A -85,B 0,C 180,E1 -20279.438,E2 -20279.438} C_VEL
LIN {X 0,Y 243.18,Z 490.161,A -85,B 0,C 180,E1 -20281.104,E2 -20281.104} C_VEL
LIN {X 0,Y 246.238,Z 481.47,A -85,B 0,C 180,E1 -20282.355,E2 -20282.355} C_VEL
LIN {X 0,Y 248.926,Z 472.648,A -85,B 0,C 180,E1 -20283.405,E2 -20283.405} C_VEL
LIN {X 0,Y 251.606,Z 462.649,A -85,B 0,C 180,E1 -20284.325,E2 -20284.325} C_VEL
LIN {X 0,Y 253.916,Z 452.212,A -85,B 0,C 180,E1 -20285.052,E2 -20285.052} C_VEL
LIN {X 0,Y 255.699,Z 441.766,A -85,B 0,C 180,E1 -20285.586,E2 -20285.586} C_VEL
LIN {X 0,Y 261.333,Z 391.022,A -85,B 0,C 180,E1 -20287.608,E2 -20287.608} C_VEL
LIN {X 0,Y 261.084,Z 384.458,A -85,B 0,C 180,E1 -20288.217,E2 -20288.217} C_VEL
LIN {X 0,Y 258.135,Z 377.279,A -85,B 0,C 180,E1 -20289.913,E2 -20289.913} C_VEL
LIN {X 0,Y 255.184,Z 370.981,A -85,B 0,C 180,E1 -20291.792,E2 -20291.792} C_VEL
LIN {X 0,Y 252.194,Z 365.457,A -85,B 0,C 180,E1 -20293.947,E2 -20293.947} C_VEL
LIN {X 0,Y 249.296,Z 360.433,A -85,B 0,C 180,E1 -20296.479,E2 -20296.479} C_VEL
LIN {X 0,Y 246.012,Z 355.365,A -85,B 0,C 180,E1 -20300.472,E2 -20300.472} C_VEL
LIN {X 0,Y 244.747,Z 353.376,A -85,B 0,C 180,E1 -20303.224,E2 -20303.224} C_VEL
LIN {X 0,Y 244.352,Z 352.861,A -85,B 0,C 180,E1 -20304.885,E2 -20304.885} C_VEL
LIN {X 0,Y 244.473,Z 352.919,A -85,B 0,C 180,E1 -20308.839,E2 -20308.839} C_VEL
LIN {X 0,Y 245.89,Z 354.404,A -85,B 0,C 180,E1 -20312.251,E2 -20312.251} C_VEL
LIN {X 0,Y 249.389,Z 359.547,A -85,B 0,C 180,E1 -20316.611,E2 -20316.611} C_VEL
LIN {X 0,Y 253.094,Z 365.591,A -85,B 0,C 180,E1 -20319.769,E2 -20319.769} C_VEL
LIN {X 0,Y 256.022,Z 370.968,A -85,B 0,C 180,E1 -20321.825,E2 -20321.825} C_VEL
LIN {X 0,Y 259.187,Z 377.611,A -85,B 0,C 180,E1 -20323.822,E2 -20323.822} C_VEL
LIN {X 0,Y 260.481,Z 380.973,A -85,B 0,C 180,E1 -20324.599,E2 -20324.599} C_VEL
LIN {X 0,Y 260.855,Z 389.881,A -85,B 0,C 180,E1 -20325.513,E2 -20325.513} C_VEL
LIN {X 0,Y 255.347,Z 433.678,A -85,B 0,C 180,E1 -20327.483,E2 -20327.483} C_VEL
LIN {X 0,Y 253.155,Z 446.147,A -85,B 0,C 180,E1 -20328.288,E2 -20328.288} C_VEL
LIN {X 0,Y 250.616,Z 457.01,A -85,B 0,C 180,E1 -20329.295,E2 -20329.295} C_VEL
LIN {X 0,Y 247.929,Z 466.474,A -85,B 0,C 180,E1 -20330.414,E2 -20330.414} C_VEL
LIN {X 0,Y 244.973,Z 475.447,A -85,B 0,C 180,E1 -20331.754,E2 -20331.754} C_VEL
LIN {X 0,Y 241.734,Z 483.966,A -85,B 0,C 180,E1 -20333.323,E2 -20333.323} C_VEL
LIN {X 0,Y 237.978,Z 492.732,A -85,B 0,C 180,E1 -20335.343,E2 -20335.343} C_VEL
LIN {X 0,Y 234.533,Z 499.638,A -85,B 0,C 180,E1 -20337.425,E2 -20337.425} C_VEL
LIN {X 0,Y 231.454,Z 505.11,A -85,B 0,C 180,E1 -20339.521,E2 -20339.521} C_VEL
LIN {X 0,Y 228.603,Z 509.661,A -85,B 0,C 180,E1 -20341.763,E2 -20341.763} C_VEL
LIN {X 0,Y 226.656,Z 512.531,A -85,B 0,C 180,E1 -20343.556,E2 -20343.556} C_VEL
LIN {X 0,Y 224.963,Z 514.779,A -85,B 0,C 180,E1 -20345.379,E2 -20345.379} C_VEL
LIN {X 0,Y 223.434,Z 516.367,A -85,B 0,C 180,E1 -20347.229,E2 -20347.229} C_VEL
LIN {X 0,Y 221.423,Z 517.93,A -85,B 0,C 180,E1 -20350.292,E2 -20350.292} C_VEL
LIN {X 0,Y 220.161,Z 518.099,A -85,B 0,C 180,E1 -20352.913,E2 -20352.913} C_VEL
LIN {X 0,Y 219.191,Z 517.027,A -85,B 0,C 180,E1 -20355.873,E2 -20355.873} C_VEL
LIN {X 0,Y 218.613,Z 513.767,A -85,B 0,C 180,E1 -20359.729,E2 -20359.729} C_VEL
LIN {X 0,Y 218.657,Z 509.707,A -85,B 0,C 180,E1 -20362.688,E2 -20362.688} C_VEL
LIN {X 0,Y 219.015,Z 504.523,A -85,B 0,C 180,E1 -20365.38,E2 -20365.38} C_VEL
LIN {X 0,Y 219.419,Z 498.927,A -85,B 0,C 180,E1 -20367.675,E2 -20367.675} C_VEL
LIN {X 0,Y 220.057,Z 491.645,A -85,B 0,C 180,E1 -20370.077,E2 -20370.077} C_VEL
LIN {X 0,Y 220.927,Z 482.632,A -85,B 0,C 180,E1 -20372.468,E2 -20372.468} C_VEL
LIN {X 0,Y 221.935,Z 472.342,A -85,B 0,C 180,E1 -20374.581,E2 -20374.581} C_VEL
LIN {X 0,Y 222.694,Z 463.85,A -85,B 0,C 180,E1 -20376.001,E2 -20376.001} C_VEL
LIN {X 0,Y 223.482,Z 454.678,A -85,B 0,C 180,E1 -20377.257,E2 -20377.257} C_VEL
LIN {X 0,Y 224.249,Z 445.135,A -85,B 0,C 180,E1 -20378.302,E2 -20378.302} C_VEL
LIN {X 0,Y 224.996,Z 431.935,A -85,B 0,C 180,E1 -20379.383,E2 -20379.383} C_VEL
LIN {X 0,Y 226.009,Z 409.999,A -85,B 0,C 180,E1 -20380.477,E2 -20380.477} C_VEL
LIN {X 0,Y 227.341,Z 374.687,A -85,B 0,C 180,E1 -20382.105,E2 -20382.105} C_VEL
LIN {X 0,Y 224.027,Z 340.87,A -85,B 0,C 180,E1 -20383.917,E2 -20383.917} C_VEL
LIN {X 0,Y 224.954,Z 335.002,A -85,B 0,C 180,E1 -20385.938,E2 -20385.938} C_VEL
LIN {X 0,Y 224.637,Z 331.825,A -85,B 0,C 180,E1 -20387.12,E2 -20387.12} C_VEL
LIN {X 0,Y 222.532,Z 321.113,A -85,B 0,C 180,E1 -20391.31,E2 -20391.31} C_VEL
LIN {X 0,Y 220.857,Z 312.97,A -85,B 0,C 180,E1 -20394.707,E2 -20394.707} C_VEL
LIN {X 0,Y 220.839,Z 312.975,A -85,B 0,C 180,E1 -20399.39,E2 -20399.39} C_VEL
LIN {X 0,Y 220.834,Z 312.976,A -85,B 0,C 180,E1 -20403.54,E2 -20403.54} C_VEL
LIN {X 0,Y 220.86,Z 312.972,A -85,B 0,C 180,E1 -20407.55,E2 -20407.55} C_VEL
LIN {X 0,Y 220.927,Z 312.967,A -85,B 0,C 180,E1 -20412.623,E2 -20412.623} C_VEL
LIN {X 0,Y 220.992,Z 312.956,A -85,B 0,C 180,E1 -20417.135,E2 -20417.135} C_VEL
LIN {X 0,Y 221.2,Z 312.931,A -85,B 0,C 180,E1 -20420.856,E2 -20420.856} C_VEL
LIN {X 0,Y 221.243,Z 312.924,A -85,B 0,C 180,E1 -20422.697,E2 -20422.697} C_VEL
LIN {X 0,Y 221.469,Z 312.896,A -85,B 0,C 180,E1 -20428.178,E2 -20428.178} C_VEL
LIN {X 0,Y 221.468,Z 312.898,A -85,B 0,C 180,E1 -20431.815,E2 -20431.815} C_VEL
LIN {X 0,Y 221.245,Z 312.923,A -85,B 0,C 180,E1 -20437.295,E2 -20437.295} C_VEL
LIN {X 0,Y 221.066,Z 312.944,A -85,B 0,C 180,E1 -20440.992,E2 -20440.992} C_VEL
LIN {X 0,Y 220.968,Z 312.961,A -85,B 0,C 180,E1 -20444.735,E2 -20444.735} C_VEL
LIN {X 0,Y 220.867,Z 312.973,A -85,B 0,C 180,E1 -20448.548,E2 -20448.548} C_VEL
LIN {X 0,Y 220.838,Z 312.972,A -85,B 0,C 180,E1 -20452.643,E2 -20452.643} C_VEL
LIN {X 0,Y 220.857,Z 312.974,A -85,B 0,C 180,E1 -20456.998,E2 -20456.998} C_VEL
LIN {X 0,Y 220.809,Z 312.974,A -85,B 0,C 180,E1 -20460.752,E2 -20460.752} C_VEL
LIN {X 0,Y 220.781,Z 312.981,A -85,B 0,C 180,E1 -20464.95,E2 -20464.95} C_VEL
LIN {X 0,Y 220.787,Z 312.98,A -85,B 0,C 180,E1 -20467.269,E2 -20467.269} C_VEL
LIN {X 0,Y 220.745,Z 312.987,A -85,B 0,C 180,E1 -20471.948,E2 -20471.948} C_VEL
LIN {X 0,Y 220.746,Z 312.985,A -85,B 0,C 180,E1 -20475.538,E2 -20475.538} C_VEL
LIN {X 0,Y 220.762,Z 312.984,A -85,B 0,C 180,E1 -20480.452,E2 -20480.452} C_VEL
LIN {X 0,Y 220.802,Z 312.983,A -85,B 0,C 180,E1 -20482.787,E2 -20482.787} C_VEL
LIN {X 0,Y 220.791,Z 312.98,A -85,B 0,C 180,E1 -20487.238,E2 -20487.238} C_VEL
LIN {X 0,Y 220.807,Z 312.981,A -85,B 0,C 180,E1 -20491.481,E2 -20491.481} C_VEL
LIN {X 0,Y 220.828,Z 312.975,A -85,B 0,C 180,E1 -20495.559,E2 -20495.559} C_VEL
LIN {X 0,Y 220.813,Z 312.979,A -85,B 0,C 180,E1 -20499.505,E2 -20499.505} C_VEL
LIN {X 0,Y 220.941,Z 312.961,A -85,B 0,C 180,E1 -20503.363,E2 -20503.363} C_VEL
LIN {X 0,Y 221.025,Z 312.951,A -85,B 0,C 180,E1 -20509,E2 -20509} C_VEL
LIN {X 0,Y 221.214,Z 312.927,A -85,B 0,C 180,E1 -20512.698,E2 -20512.698} C_VEL
LIN {X 0,Y 221.475,Z 312.895,A -85,B 0,C 180,E1 -20518.181,E2 -20518.181} C_VEL
LIN {X 0,Y 221.47,Z 312.893,A -85,B 0,C 180,E1 -20521.818,E2 -20521.818} C_VEL
LIN {X 0,Y 221.216,Z 312.931,A -85,B 0,C 180,E1 -20527.3,E2 -20527.3} C_VEL
LIN {X 0,Y 221.025,Z 312.95,A -85,B 0,C 180,E1 -20530.998,E2 -20530.998} C_VEL
LIN {X 0,Y 220.971,Z 312.958,A -85,B 0,C 180,E1 -20536.632,E2 -20536.632} C_VEL
LIN {X 0,Y 220.846,Z 312.971,A -85,B 0,C 180,E1 -20540.49,E2 -20540.49} C_VEL
LIN {X 0,Y 220.822,Z 312.979,A -85,B 0,C 180,E1 -20544.439,E2 -20544.439} C_VEL
LIN {X 0,Y 220.778,Z 312.982,A -85,B 0,C 180,E1 -20548.521,E2 -20548.521} C_VEL
LIN {X 0,Y 220.781,Z 312.985,A -85,B 0,C 180,E1 -20552.761,E2 -20552.761} C_VEL
LIN {X 0,Y 220.773,Z 312.986,A -85,B 0,C 180,E1 -20557.279,E2 -20557.279} C_VEL
LIN {X 0,Y 220.734,Z 312.988,A -85,B 0,C 180,E1 -20561.96,E2 -20561.96} C_VEL
LIN {X 0,Y 220.742,Z 312.99,A -85,B 0,C 180,E1 -20565.549,E2 -20565.549} C_VEL
LIN {X 0,Y 220.786,Z 312.983,A -85,B 0,C 180,E1 -20570.468,E2 -20570.468} C_VEL
LIN {X 0,Y 220.888,Z 313.083,A -85,B 0,C 180,E1 -20571.995,E2 -20571.995} C_VEL
LIN {X 0,Y 221.174,Z 314.505,A -85,B 0,C 180,E1 -20572.528,E2 -20572.528} C_VEL
LIN {X 0,Y 221.248,Z 318.008,A -85,B 0,C 180,E1 -20573.759,E2 -20573.759} C_VEL
LIN {X 0,Y 219.687,Z 324.151,A -85,B 0,C 180,E1 -20575.74,E2 -20575.74} C_VEL
LIN {X 0,Y 218.302,Z 329.131,A -85,B 0,C 180,E1 -20577.337,E2 -20577.337} C_VEL
LIN {X 0,Y 218.015,Z 332.791,A -85,B 0,C 180,E1 -20578.571,E2 -20578.571} C_VEL
LIN {X 0,Y 218.171,Z 333.976,A -85,B 0,C 180,E1 -20578.988,E2 -20578.988} C_VEL
LIN {X 0,Y 219.486,Z 340.544,A -85,B 0,C 180,E1 -20581.302,E2 -20581.302} C_VEL
LIN {X 0,Y 219.323,Z 343.42,A -85,B 0,C 180,E1 -20582.256,E2 -20582.256} C_VEL
LIN {X 0,Y 219.225,Z 343.803,A -85,B 0,C 180,E1 -20582.379,E2 -20582.379} C_VEL
LIN {X 0,Y 220.35,Z 365.489,A -85,B 0,C 180,E1 -20583.429,E2 -20583.429} C_VEL
LIN {X 0,Y 221.652,Z 382.875,A -85,B 0,C 180,E1 -20584.286,E2 -20584.286} C_VEL
LIN {X 0,Y 219.328,Z 443.815,A -85,B 0,C 180,E1 -20586.957,E2 -20586.957} C_VEL
LIN {X 0,Y 218.701,Z 454.245,A -85,B 0,C 180,E1 -20587.635,E2 -20587.635} C_VEL
LIN {X 0,Y 217.898,Z 463.828,A -85,B 0,C 180,E1 -20588.483,E2 -20588.483} C_VEL
LIN {X 0,Y 217.034,Z 473.602,A -85,B 0,C 180,E1 -20589.596,E2 -20589.596} C_VEL
LIN {X 0,Y 216.222,Z 481.631,A -85,B 0,C 180,E1 -20590.718,E2 -20590.718} C_VEL
LIN {X 0,Y 215.278,Z 490.32,A -85,B 0,C 180,E1 -20592.184,E2 -20592.184} C_VEL
LIN {X 0,Y 214.366,Z 498.411,A -85,B 0,C 180,E1 -20593.825,E2 -20593.825} C_VEL
LIN {X 0,Y 213.515,Z 506.179,A -85,B 0,C 180,E1 -20595.713,E2 -20595.713} C_VEL
LIN {X 0,Y 212.933,Z 512.783,A -85,B 0,C 180,E1 -20597.617,E2 -20597.617} C_VEL
LIN {X 0,Y 212.438,Z 519.627,A -85,B 0,C 180,E1 -20600.003,E2 -20600.003} C_VEL
LIN {X 0,Y 212.166,Z 525.235,A -85,B 0,C 180,E1 -20602.391,E2 -20602.391} C_VEL
LIN {X 0,Y 212.122,Z 529.028,A -85,B 0,C 180,E1 -20604.3,E2 -20604.3} C_VEL
LIN {X 0,Y 212.017,Z 533.387,A -85,B 0,C 180,E1 -20607.154,E2 -20607.154} C_VEL
LIN {X 0,Y 212.247,Z 536.554,A -85,B 0,C 180,E1 -20610.004,E2 -20610.004} C_VEL
LIN {X 0,Y 211.789,Z 537.992,A -85,B 0,C 180,E1 -20611.905,E2 -20611.905} C_VEL
LIN {X 0,Y 211.625,Z 539.407,A -85,B 0,C 180,E1 -20614.949,E2 -20614.949} C_VEL
LIN {X 0,Y 211.694,Z 539.707,A -85,B 0,C 180,E1 -20617.634,E2 -20617.634} C_VEL
LIN {X 0,Y 212.466,Z 538.824,A -85,B 0,C 180,E1 -20621.45,E2 -20621.45} C_VEL
LIN {X 0,Y 214.167,Z 536.203,A -85,B 0,C 180,E1 -20625.222,E2 -20625.222} C_VEL
LIN {X 0,Y 216.243,Z 533.172,A -85,B 0,C 180,E1 -20627.986,E2 -20627.986} C_VEL
LIN {X 0,Y 218.657,Z 529.103,A -85,B 0,C 180,E1 -20630.707,E2 -20630.707} C_VEL
LIN {X 0,Y 220.57,Z 525.888,A -85,B 0,C 180,E1 -20632.481,E2 -20632.481} C_VEL
LIN {X 0,Y 224.064,Z 519.848,A -85,B 0,C 180,E1 -20635.053,E2 -20635.053} C_VEL
LIN {X 0,Y 227.473,Z 513.726,A -85,B 0,C 180,E1 -20637.112,E2 -20637.112} C_VEL
LIN {X 0,Y 231.089,Z 506.389,A -85,B 0,C 180,E1 -20639.118,E2 -20639.118} C_VEL
LIN {X 0,Y 234.337,Z 499.566,A -85,B 0,C 180,E1 -20640.654,E2 -20640.654} C_VEL
LIN {X 0,Y 238.195,Z 490.364,A -85,B 0,C 180,E1 -20642.329,E2 -20642.329} C_VEL
LIN {X 0,Y 241.41,Z 481.813,A -85,B 0,C 180,E1 -20643.582,E2 -20643.582} C_VEL
LIN {X 0,Y 244.231,Z 473.122,A -85,B 0,C 180,E1 -20644.634,E2 -20644.634} C_VEL
LIN {X 0,Y 247.016,Z 463.316,A -85,B 0,C 180,E1 -20645.555,E2 -20645.555} C_VEL
LIN {X 0,Y 249.706,Z 451.93,A -85,B 0,C 180,E1 -20646.356,E2 -20646.356} C_VEL
LIN {X 0,Y 251.602,Z 441.339,A -85,B 0,C 180,E1 -20646.91,E2 -20646.91} C_VEL
LIN {X 0,Y 257.4,Z 392.236,A -85,B 0,C 180,E1 -20648.901,E2 -20648.901} C_VEL
LIN {X 0,Y 257.253,Z 388.295,A -85,B 0,C 180,E1 -20649.286,E2 -20649.286} C_VEL
LIN {X 0,Y 254.4,Z 380.866,A -85,B 0,C 180,E1 -20651.165,E2 -20651.165} C_VEL
LIN {X 0,Y 251.643,Z 375.216,A -85,B 0,C 180,E1 -20653.093,E2 -20653.093} C_VEL
LIN {X 0,Y 249.852,Z 371.667,A -85,B 0,C 180,E1 -20654.518,E2 -20654.518} C_VEL
LIN {X 0,Y 247.251,Z 366.899,A -85,B 0,C 180,E1 -20656.986,E2 -20656.986} C_VEL
LIN {X 0,Y 244.213,Z 361.748,A -85,B 0,C 180,E1 -20661.116,E2 -20661.116} C_VEL
LIN {X 0,Y 243.073,Z 359.967,A -85,B 0,C 180,E1 -20664.051,E2 -20664.051} C_VEL
LIN {X 0,Y 242.742,Z 359.7,A -85,B 0,C 180,E1 -20667.098,E2 -20667.098} C_VEL
LIN {X 0,Y 243.526,Z 360.349,A -85,B 0,C 180,E1 -20670.383,E2 -20670.383} C_VEL
LIN {X 0,Y 244.499,Z 361.669,A -85,B 0,C 180,E1 -20672.461,E2 -20672.461} C_VEL
LIN {X 0,Y 247.693,Z 366.665,A -85,B 0,C 180,E1 -20676.518,E2 -20676.518} C_VEL
LIN {X 0,Y 250.74,Z 371.966,A -85,B 0,C 180,E1 -20679.274,E2 -20679.274} C_VEL
LIN {X 0,Y 253.313,Z 377.041,A -85,B 0,C 180,E1 -20681.246,E2 -20681.246} C_VEL
LIN {X 0,Y 256.128,Z 383.269,A -85,B 0,C 180,E1 -20683.14,E2 -20683.14} C_VEL
LIN {X 0,Y 256.753,Z 385.319,A -85,B 0,C 180,E1 -20683.607,E2 -20683.607} C_VEL
LIN {X 0,Y 256.858,Z 392.089,A -85,B 0,C 180,E1 -20684.281,E2 -20684.281} C_VEL
LIN {X 0,Y 251.332,Z 433.709,A -85,B 0,C 180,E1 -20686.148,E2 -20686.148} C_VEL
LIN {X 0,Y 249.039,Z 446.123,A -85,B 0,C 180,E1 -20686.953,E2 -20686.953} C_VEL
LIN {X 0,Y 246.086,Z 457.863,A -85,B 0,C 180,E1 -20688.051,E2 -20688.051} C_VEL
LIN {X 0,Y 243.283,Z 467.126,A -85,B 0,C 180,E1 -20689.16,E2 -20689.16} C_VEL
LIN {X 0,Y 240.132,Z 476.197,A -85,B 0,C 180,E1 -20690.525,E2 -20690.525} C_VEL
LIN {X 0,Y 237.128,Z 483.672,A -85,B 0,C 180,E1 -20691.908,E2 -20691.908} C_VEL
LIN {X 0,Y 233.254,Z 492.169,A -85,B 0,C 180,E1 -20693.857,E2 -20693.857} C_VEL
LIN {X 0,Y 229.371,Z 499.58,A -85,B 0,C 180,E1 -20696.048,E2 -20696.048} C_VEL
LIN {X 0,Y 225.96,Z 505.28,A -85,B 0,C 180,E1 -20698.219,E2 -20698.219} C_VEL
LIN {X 0,Y 223.51,Z 509.044,A -85,B 0,C 180,E1 -20700.001,E2 -20700.001} C_VEL
LIN {X 0,Y 220.267,Z 513.304,A -85,B 0,C 180,E1 -20702.744,E2 -20702.744} C_VEL
LIN {X 0,Y 218.542,Z 515.402,A -85,B 0,C 180,E1 -20704.527,E2 -20704.527} C_VEL
LIN {X 0,Y 216.096,Z 517.6,A -85,B 0,C 180,E1 -20707.476,E2 -20707.476} C_VEL
LIN {X 0,Y 214.274,Z 518.504,A -85,B 0,C 180,E1 -20710.282,E2 -20710.282} C_VEL
LIN {X 0,Y 212.849,Z 518.238,A -85,B 0,C 180,E1 -20713.365,E2 -20713.365} C_VEL
LIN {X 0,Y 212.061,Z 516.973,A -85,B 0,C 180,E1 -20716.04,E2 -20716.04} C_VEL
LIN {X 0,Y 211.61,Z 515.042,A -85,B 0,C 180,E1 -20718.393,E2 -20718.393} C_VEL
LIN {X 0,Y 211.512,Z 512.759,A -85,B 0,C 180,E1 -20720.42,E2 -20720.42} C_VEL
LIN {X 0,Y 211.56,Z 509.847,A -85,B 0,C 180,E1 -20722.459,E2 -20722.459} C_VEL
LIN {X 0,Y 211.878,Z 505.105,A -85,B 0,C 180,E1 -20725.02,E2 -20725.02} C_VEL
LIN {X 0,Y 212.182,Z 500.667,A -85,B 0,C 180,E1 -20726.985,E2 -20726.985} C_VEL
LIN {X 0,Y 212.687,Z 494.617,A -85,B 0,C 180,E1 -20729.171,E2 -20729.171} C_VEL
LIN {X 0,Y 213.343,Z 487.37,A -85,B 0,C 180,E1 -20731.313,E2 -20731.313} C_VEL
LIN {X 0,Y 214.203,Z 479.016,A -85,B 0,C 180,E1 -20733.339,E2 -20733.339} C_VEL
LIN {X 0,Y 215.023,Z 470.317,A -85,B 0,C 180,E1 -20735.072,E2 -20735.072} C_VEL
LIN {X 0,Y 215.971,Z 460.136,A -85,B 0,C 180,E1 -20736.724,E2 -20736.724} C_VEL
LIN {X 0,Y 216.957,Z 447.996,A -85,B 0,C 180,E1 -20738.217,E2 -20738.217} C_VEL
LIN {X 0,Y 217.625,Z 437.512,A -85,B 0,C 180,E1 -20739.191,E2 -20739.191} C_VEL
LIN {X 0,Y 218.259,Z 426.333,A -85,B 0,C 180,E1 -20739.943,E2 -20739.943} C_VEL
LIN {X 0,Y 220.359,Z 375.217,A -85,B 0,C 180,E1 -20742.43,E2 -20742.43} C_VEL
LIN {X 0,Y 217.081,Z 340.892,A -85,B 0,C 180,E1 -20744.323,E2 -20744.323} C_VEL
LIN {X 0,Y 217.946,Z 335.109,A -85,B 0,C 180,E1 -20746.399,E2 -20746.399} C_VEL
LIN {X 0,Y 216.527,Z 327.204,A -85,B 0,C 180,E1 -20749.522,E2 -20749.522} C_VEL
LIN {X 0,Y 214.408,Z 316.735,A -85,B 0,C 180,E1 -20753.841,E2 -20753.841} C_VEL
LIN {X 0,Y 213.828,Z 313.847,A -85,B 0,C 180,E1 -20755.132,E2 -20755.132} C_VEL
LIN {X 0,Y 213.773,Z 313.855,A -85,B 0,C 180,E1 -20758.737,E2 -20758.737} C_VEL
LIN {X 0,Y 213.771,Z 313.857,A -85,B 0,C 180,E1 -20762.594,E2 -20762.594} C_VEL
LIN {X 0,Y 213.8,Z 313.852,A -85,B 0,C 180,E1 -20766.989,E2 -20766.989} C_VEL
LIN {X 0,Y 213.891,Z 313.843,A -85,B 0,C 180,E1 -20772.797,E2 -20772.797} C_VEL
LIN {X 0,Y 213.93,Z 313.833,A -85,B 0,C 180,E1 -20776.703,E2 -20776.703} C_VEL
LIN {X 0,Y 214.14,Z 313.809,A -85,B 0,C 180,E1 -20780.552,E2 -20780.552} C_VEL
LIN {X 0,Y 214.074,Z 313.813,A -85,B 0,C 180,E1 -20784.345,E2 -20784.345} C_VEL
LIN {X 0,Y 214.405,Z 313.776,A -85,B 0,C 180,E1 -20788.118,E2 -20788.118} C_VEL
LIN {X 0,Y 214.516,Z 313.764,A -85,B 0,C 180,E1 -20789.996,E2 -20789.996} C_VEL
LIN {X 0,Y 214.405,Z 313.777,A -85,B 0,C 180,E1 -20791.874,E2 -20791.874} C_VEL
LIN {X 0,Y 214.186,Z 313.803,A -85,B 0,C 180,E1 -20797.537,E2 -20797.537} C_VEL
LIN {X 0,Y 213.997,Z 313.824,A -85,B 0,C 180,E1 -20801.359,E2 -20801.359} C_VEL
LIN {X 0,Y 213.902,Z 313.838,A -85,B 0,C 180,E1 -20805.234,E2 -20805.234} C_VEL
LIN {X 0,Y 213.793,Z 313.852,A -85,B 0,C 180,E1 -20809.186,E2 -20809.186} C_VEL
LIN {X 0,Y 213.789,Z 313.854,A -85,B 0,C 180,E1 -20813.227,E2 -20813.227} C_VEL
LIN {X 0,Y 213.778,Z 313.856,A -85,B 0,C 180,E1 -20817.421,E2 -20817.421} C_VEL
LIN {X 0,Y 213.748,Z 313.859,A -85,B 0,C 180,E1 -20821.733,E2 -20821.733} C_VEL
LIN {X 0,Y 213.728,Z 313.86,A -85,B 0,C 180,E1 -20826.282,E2 -20826.282} C_VEL
LIN {X 0,Y 213.688,Z 313.863,A -85,B 0,C 180,E1 -20831.121,E2 -20831.121} C_VEL
LIN {X 0,Y 213.685,Z 313.866,A -85,B 0,C 180,E1 -20833.673,E2 -20833.673} C_VEL
LIN {X 0,Y 213.684,Z 313.868,A -85,B 0,C 180,E1 -20836.339,E2 -20836.339} C_VEL
LIN {X 0,Y 213.686,Z 313.863,A -85,B 0,C 180,E1 -20839.14,E2 -20839.14} C_VEL
LIN {X 0,Y 213.717,Z 313.861,A -85,B 0,C 180,E1 -20843.705,E2 -20843.705} C_VEL
LIN {X 0,Y 213.755,Z 313.855,A -85,B 0,C 180,E1 -20848.726,E2 -20848.726} C_VEL
LIN {X 0,Y 213.799,Z 313.851,A -85,B 0,C 180,E1 -20852.598,E2 -20852.598} C_VEL
LIN {X 0,Y 213.769,Z 313.852,A -85,B 0,C 180,E1 -20856.982,E2 -20856.982} C_VEL
LIN {X 0,Y 213.849,Z 313.844,A -85,B 0,C 180,E1 -20862.795,E2 -20862.795} C_VEL
LIN {X 0,Y 213.887,Z 313.839,A -85,B 0,C 180,E1 -20866.701,E2 -20866.701} C_VEL
LIN {X 0,Y 214.091,Z 313.817,A -85,B 0,C 180,E1 -20870.552,E2 -20870.552} C_VEL
LIN {X 0,Y 214.06,Z 313.817,A -85,B 0,C 180,E1 -20874.346,E2 -20874.346} C_VEL
LIN {X 0,Y 214.408,Z 313.775,A -85,B 0,C 180,E1 -20878.121,E2 -20878.121} C_VEL
LIN {X 0,Y 214.505,Z 313.763,A -85,B 0,C 180,E1 -20879.999,E2 -20879.999} C_VEL
LIN {X 0,Y 214.403,Z 313.773,A -85,B 0,C 180,E1 -20881.877,E2 -20881.877} C_VEL
LIN {X 0,Y 214.156,Z 313.809,A -85,B 0,C 180,E1 -20887.542,E2 -20887.542} C_VEL
LIN {X 0,Y 213.957,Z 313.831,A -85,B 0,C 180,E1 -20891.366,E2 -20891.366} C_VEL
LIN {X 0,Y 213.879,Z 313.841,A -85,B 0,C 180,E1 -20895.24,E2 -20895.24} C_VEL
LIN {X 0,Y 213.798,Z 313.85,A -85,B 0,C 180,E1 -20899.19,E2 -20899.19} C_VEL
LIN {X 0,Y 213.77,Z 313.854,A -85,B 0,C 180,E1 -20903.235,E2 -20903.235} C_VEL
LIN {X 0,Y 213.762,Z 313.854,A -85,B 0,C 180,E1 -20907.434,E2 -20907.434} C_VEL
LIN {X 0,Y 213.728,Z 313.859,A -85,B 0,C 180,E1 -20911.743,E2 -20911.743} C_VEL
LIN {X 0,Y 213.713,Z 313.861,A -85,B 0,C 180,E1 -20916.293,E2 -20916.293} C_VEL
LIN {X 0,Y 213.678,Z 313.871,A -85,B 0,C 180,E1 -20921.132,E2 -20921.132} C_VEL
LIN {X 0,Y 213.679,Z 313.869,A -85,B 0,C 180,E1 -20923.684,E2 -20923.684} C_VEL
LIN {X 0,Y 213.68,Z 313.867,A -85,B 0,C 180,E1 -20926.35,E2 -20926.35} C_VEL
LIN {X 0,Y 213.768,Z 313.865,A -85,B 0,C 180,E1 -20931.461,E2 -20931.461} C_VEL
LIN {X 0,Y 216.37,Z 325.569,A -85,B 0,C 180,E1 -20935.932,E2 -20935.932} C_VEL
LIN {X 0,Y 218.171,Z 333.976,A -85,B 0,C 180,E1 -20938.988,E2 -20938.988} C_VEL
LIN {X 0,Y 217.896,Z 336.515,A -85,B 0,C 180,E1 -20939.827,E2 -20939.827} C_VEL
LIN {X 0,Y 216.056,Z 340.157,A -85,B 0,C 180,E1 -20940.82,E2 -20940.82} C_VEL
LIN {X 0,Y 213.83,Z 344.233,A -85,B 0,C 180,E1 -20941.628,E2 -20941.628} C_VEL
LIN {X 0,Y 212.544,Z 348.401,A -85,B 0,C 180,E1 -20942.139,E2 -20942.139} C_VEL
LIN {X 0,Y 212.447,Z 350.36,A -85,B 0,C 180,E1 -20942.275,E2 -20942.275} C_VEL
LIN {X 0,Y 214.664,Z 383.334,A -85,B 0,C 180,E1 -20943.963,E2 -20943.963} C_VEL
LIN {X 0,Y 212.291,Z 444.001,A -85,B 0,C 180,E1 -20946.728,E2 -20946.728} C_VEL
LIN {X 0,Y 211.656,Z 454.27,A -85,B 0,C 180,E1 -20947.429,E2 -20947.429} C_VEL
LIN {X 0,Y 210.797,Z 464.333,A -85,B 0,C 180,E1 -20948.363,E2 -20948.363} C_VEL
LIN {X 0,Y 209.958,Z 473.453,A -85,B 0,C 180,E1 -20949.45,E2 -20949.45} C_VEL
LIN {X 0,Y 209.136,Z 481.544,A -85,B 0,C 180,E1 -20950.625,E2 -20950.625} C_VEL
LIN {X 0,Y 208.22,Z 489.822,A -85,B 0,C 180,E1 -20952.068,E2 -20952.068} C_VEL
LIN {X 0,Y 207.287,Z 497.934,A -85,B 0,C 180,E1 -20953.763,E2 -20953.763} C_VEL
LIN {X 0,Y 206.43,Z 505.706,A -85,B 0,C 180,E1 -20955.716,E2 -20955.716} C_VEL
LIN {X 0,Y 205.845,Z 512.302,A -85,B 0,C 180,E1 -20957.684,E2 -20957.684} C_VEL
LIN {X 0,Y 205.374,Z 519.14,A -85,B 0,C 180,E1 -20960.153,E2 -20960.153} C_VEL
LIN {X 0,Y 205.163,Z 523.777,A -85,B 0,C 180,E1 -20962.129,E2 -20962.129} C_VEL
LIN {X 0,Y 205.073,Z 529.289,A -85,B 0,C 180,E1 -20965.09,E2 -20965.09} C_VEL
LIN {X 0,Y 205.006,Z 533.446,A -85,B 0,C 180,E1 -20968.04,E2 -20968.04} C_VEL
LIN {X 0,Y 205.193,Z 535.655,A -85,B 0,C 180,E1 -20970.004,E2 -20970.004} C_VEL
LIN {X 0,Y 204.681,Z 538.251,A -85,B 0,C 180,E1 -20973.941,E2 -20973.941} C_VEL
LIN {X 0,Y 204.553,Z 539.006,A -85,B 0,C 180,E1 -20975.92,E2 -20975.92} C_VEL
LIN {X 0,Y 204.955,Z 539.066,A -85,B 0,C 180,E1 -20979.875,E2 -20979.875} C_VEL
LIN {X 0,Y 205.476,Z 538.557,A -85,B 0,C 180,E1 -20981.845,E2 -20981.845} C_VEL
LIN {X 0,Y 207.32,Z 536.238,A -85,B 0,C 180,E1 -20985.738,E2 -20985.738} C_VEL
LIN {X 0,Y 209.504,Z 533.425,A -85,B 0,C 180,E1 -20988.586,E2 -20988.586} C_VEL
LIN {X 0,Y 212.034,Z 529.619,A -85,B 0,C 180,E1 -20991.385,E2 -20991.385} C_VEL
LIN {X 0,Y 215.278,Z 524.682,A -85,B 0,C 180,E1 -20994.086,E2 -20994.086} C_VEL
LIN {X 0,Y 219.049,Z 518.485,A -85,B 0,C 180,E1 -20996.692,E2 -20996.692} C_VEL
LIN {X 0,Y 222.68,Z 512.276,A -85,B 0,C 180,E1 -20998.772,E2 -20998.772} C_VEL
LIN {X 0,Y 226.676,Z 504.819,A -85,B 0,C 180,E1 -21000.77,E2 -21000.77} C_VEL
LIN {X 0,Y 230.155,Z 497.762,A -85,B 0,C 180,E1 -21002.302,E2 -21002.302} C_VEL
LIN {X 0,Y 233.787,Z 489.442,A -85,B 0,C 180,E1 -21003.789,E2 -21003.789} C_VEL
LIN {X 0,Y 237.184,Z 480.882,A -85,B 0,C 180,E1 -21005.037,E2 -21005.037} C_VEL
LIN {X 0,Y 240.184,Z 472.188,A -85,B 0,C 180,E1 -21006.077,E2 -21006.077} C_VEL
LIN {X 0,Y 243.127,Z 462.378,A -85,B 0,C 180,E1 -21006.986,E2 -21006.986} C_VEL
LIN {X 0,Y 245.651,Z 452.22,A -85,B 0,C 180,E1 -21007.7,E2 -21007.7} C_VEL
LIN {X 0,Y 247.745,Z 441.001,A -85,B 0,C 180,E1 -21008.291,E2 -21008.291} C_VEL
LIN {X 0,Y 253.696,Z 393.927,A -85,B 0,C 180,E1 -21010.214,E2 -21010.214} C_VEL
LIN {X 0,Y 253.61,Z 392.176,A -85,B 0,C 180,E1 -21010.415,E2 -21010.415} C_VEL
LIN {X 0,Y 250.989,Z 385.361,A -85,B 0,C 180,E1 -21012.28,E2 -21012.28} C_VEL
LIN {X 0,Y 248.293,Z 379.323,A -85,B 0,C 180,E1 -21014.461,E2 -21014.461} C_VEL
LIN {X 0,Y 245.24,Z 373.384,A -85,B 0,C 180,E1 -21017.47,E2 -21017.47} C_VEL
LIN {X 0,Y 242.581,Z 368.5,A -85,B 0,C 180,E1 -21021.464,E2 -21021.464} C_VEL
LIN {X 0,Y 241.547,Z 366.851,A -85,B 0,C 180,E1 -21024.416,E2 -21024.416} C_VEL
LIN {X 0,Y 241.475,Z 366.755,A -85,B 0,C 180,E1 -21028.408,E2 -21028.408} C_VEL
LIN {X 0,Y 242.606,Z 367.962,A -85,B 0,C 180,E1 -21031.624,E2 -21031.624} C_VEL
LIN {X 0,Y 245.504,Z 372.883,A -85,B 0,C 180,E1 -21035.906,E2 -21035.906} C_VEL
LIN {X 0,Y 248.35,Z 378.21,A -85,B 0,C 180,E1 -21038.723,E2 -21038.723} C_VEL
LIN {X 0,Y 250.609,Z 382.924,A -85,B 0,C 180,E1 -21040.58,E2 -21040.58} C_VEL
LIN {X 0,Y 253.036,Z 388.679,A -85,B 0,C 180,E1 -21042.368,E2 -21042.368} C_VEL
LIN {X 0,Y 253.229,Z 390.081,A -85,B 0,C 180,E1 -21042.6,E2 -21042.6} C_VEL
LIN {X 0,Y 253.176,Z 393.641,A -85,B 0,C 180,E1 -21042.948,E2 -21042.948} C_VEL
LIN {X 0,Y 247.381,Z 434.566,A -85,B 0,C 180,E1 -21044.812,E2 -21044.812} C_VEL
LIN {X 0,Y 244.805,Z 447.523,A -85,B 0,C 180,E1 -21045.665,E2 -21045.665} C_VEL
LIN {X 0,Y 241.724,Z 459.045,A -85,B 0,C 180,E1 -21046.765,E2 -21046.765} C_VEL
LIN {X 0,Y 238.742,Z 468.257,A -85,B 0,C 180,E1 -21047.894,E2 -21047.894} C_VEL
LIN {X 0,Y 235.433,Z 477.056,A -85,B 0,C 180,E1 -21049.252,E2 -21049.252} C_VEL
LIN {X 0,Y 231.808,Z 485.4,A -85,B 0,C 180,E1 -21050.842,E2 -21050.842} C_VEL
LIN {X 0,Y 227.042,Z 494.877,A -85,B 0,C 180,E1 -21053.156,E2 -21053.156} C_VEL
LIN {X 0,Y 223.608,Z 500.828,A -85,B 0,C 180,E1 -21055.043,E2 -21055.043} C_VEL
LIN {X 0,Y 220.008,Z 506.327,A -85,B 0,C 180,E1 -21057.255,E2 -21057.255} C_VEL
LIN {X 0,Y 217.266,Z 510.136,A -85,B 0,C 180,E1 -21059.176,E2 -21059.176} C_VEL
LIN {X 0,Y 215.063,Z 512.962,A -85,B 0,C 180,E1 -21060.937,E2 -21060.937} C_VEL
LIN {X 0,Y 211.989,Z 516.206,A -85,B 0,C 180,E1 -21063.803,E2 -21063.803} C_VEL
LIN {X 0,Y 210.245,Z 517.715,A -85,B 0,C 180,E1 -21065.756,E2 -21065.756} C_VEL
LIN {X 0,Y 208.713,Z 518.601,A -85,B 0,C 180,E1 -21067.742,E2 -21067.742} C_VEL
LIN {X 0,Y 207.136,Z 519.04,A -85,B 0,C 180,E1 -21070.287,E2 -21070.287} C_VEL
LIN {X 0,Y 205.556,Z 518.33,A -85,B 0,C 180,E1 -21073.848,E2 -21073.848} C_VEL
LIN {X 0,Y 204.908,Z 516.915,A -85,B 0,C 180,E1 -21076.194,E2 -21076.194} C_VEL
LIN {X 0,Y 204.472,Z 514.28,A -85,B 0,C 180,E1 -21079.059,E2 -21079.059} C_VEL
LIN {X 0,Y 204.464,Z 509.964,A -85,B 0,C 180,E1 -21082.217,E2 -21082.217} C_VEL
LIN {X 0,Y 204.762,Z 505.143,A -85,B 0,C 180,E1 -21084.864,E2 -21084.864} C_VEL
LIN {X 0,Y 205.117,Z 500.294,A -85,B 0,C 180,E1 -21087.022,E2 -21087.022} C_VEL
LIN {X 0,Y 205.595,Z 494.517,A -85,B 0,C 180,E1 -21089.153,E2 -21089.153} C_VEL
LIN {X 0,Y 206.19,Z 487.821,A -85,B 0,C 180,E1 -21091.206,E2 -21091.206} C_VEL
LIN {X 0,Y 207.003,Z 480.007,A -85,B 0,C 180,E1 -21093.194,E2 -21093.194} C_VEL
LIN {X 0,Y 207.779,Z 472.41,A -85,B 0,C 180,E1 -21094.806,E2 -21094.806} C_VEL
LIN {X 0,Y 208.563,Z 463.867,A -85,B 0,C 180,E1 -21096.309,E2 -21096.309} C_VEL
LIN {X 0,Y 209.439,Z 453.673,A -85,B 0,C 180,E1 -21097.765,E2 -21097.765} C_VEL
LIN {X 0,Y 210.414,Z 441.643,A -85,B 0,C 180,E1 -21099.084,E2 -21099.084} C_VEL
LIN {X 0,Y 211.058,Z 429.701,A -85,B 0,C 180,E1 -21099.996,E2 -21099.996} C_VEL
LIN {X 0,Y 213.347,Z 375.725,A -85,B 0,C 180,E1 -21102.753,E2 -21102.753} C_VEL
LIN {X 0,Y 210.19,Z 341.57,A -85,B 0,C 180,E1 -21104.712,E2 -21104.712} C_VEL
LIN {X 0,Y 210.171,Z 340.811,A -85,B 0,C 180,E1 -21104.772,E2 -21104.772} C_VEL
LIN {X 0,Y 210.92,Z 335.979,A -85,B 0,C 180,E1 -21106.577,E2 -21106.577} C_VEL
LIN {X 0,Y 209.225,Z 326.775,A -85,B 0,C 180,E1 -21110.34,E2 -21110.34} C_VEL
LIN {X 0,Y 207.124,Z 316.431,A -85,B 0,C 180,E1 -21114.771,E2 -21114.771} C_VEL
LIN {X 0,Y 206.758,Z 314.729,A -85,B 0,C 180,E1 -21115.59,E2 -21115.59} C_VEL
LIN {X 0,Y 206.698,Z 314.737,A -85,B 0,C 180,E1 -21119.334,E2 -21119.334} C_VEL
LIN {X 0,Y 206.677,Z 314.74,A -85,B 0,C 180,E1 -21123.763,E2 -21123.763} C_VEL
LIN {X 0,Y 206.72,Z 314.735,A -85,B 0,C 180,E1 -21128.037,E2 -21128.037} C_VEL
LIN {X 0,Y 206.828,Z 314.72,A -85,B 0,C 180,E1 -21132.19,E2 -21132.19} C_VEL
LIN {X 0,Y 206.87,Z 314.71,A -85,B 0,C 180,E1 -21136.24,E2 -21136.24} C_VEL
LIN {X 0,Y 207.085,Z 314.687,A -85,B 0,C 180,E1 -21140.227,E2 -21140.227} C_VEL
LIN {X 0,Y 207.039,Z 314.69,A -85,B 0,C 180,E1 -21144.152,E2 -21144.152} C_VEL
LIN {X 0,Y 207.345,Z 314.656,A -85,B 0,C 180,E1 -21148.054,E2 -21148.054} C_VEL
LIN {X 0,Y 207.484,Z 314.64,A -85,B 0,C 180,E1 -21149.996,E2 -21149.996} C_VEL
LIN {X 0,Y 207.345,Z 314.656,A -85,B 0,C 180,E1 -21151.938,E2 -21151.938} C_VEL
LIN {X 0,Y 207.13,Z 314.683,A -85,B 0,C 180,E1 -21157.796,E2 -21157.796} C_VEL
LIN {X 0,Y 206.92,Z 314.706,A -85,B 0,C 180,E1 -21161.753,E2 -21161.753} C_VEL
LIN {X 0,Y 206.827,Z 314.719,A -85,B 0,C 180,E1 -21165.768,E2 -21165.768} C_VEL
LIN {X 0,Y 206.713,Z 314.732,A -85,B 0,C 180,E1 -21169.87,E2 -21169.87} C_VEL
LIN {X 0,Y 206.729,Z 314.731,A -85,B 0,C 180,E1 -21174.07,E2 -21174.07} C_VEL
LIN {X 0,Y 206.68,Z 314.737,A -85,B 0,C 180,E1 -21178.421,E2 -21178.421} C_VEL
LIN {X 0,Y 206.683,Z 314.736,A -85,B 0,C 180,E1 -21182.952,E2 -21182.952} C_VEL
LIN {X 0,Y 206.655,Z 314.743,A -85,B 0,C 180,E1 -21187.736,E2 -21187.736} C_VEL
LIN {X 0,Y 206.62,Z 314.744,A -85,B 0,C 180,E1 -21191.554,E2 -21191.554} C_VEL
LIN {X 0,Y 206.612,Z 314.746,A -85,B 0,C 180,E1 -21195.576,E2 -21195.576} C_VEL
LIN {X 0,Y 206.629,Z 314.742,A -85,B 0,C 180,E1 -21199.74,E2 -21199.74} C_VEL
LIN {X 0,Y 206.676,Z 314.741,A -85,B 0,C 180,E1 -21204.683,E2 -21204.683} C_VEL
LIN {X 0,Y 206.688,Z 314.739,A -85,B 0,C 180,E1 -21209.332,E2 -21209.332} C_VEL
LIN {X 0,Y 206.701,Z 314.735,A -85,B 0,C 180,E1 -21213.767,E2 -21213.767} C_VEL
LIN {X 0,Y 206.684,Z 314.738,A -85,B 0,C 180,E1 -21218.034,E2 -21218.034} C_VEL
LIN {X 0,Y 206.772,Z 314.727,A -85,B 0,C 180,E1 -21222.186,E2 -21222.186} C_VEL
LIN {X 0,Y 206.828,Z 314.72,A -85,B 0,C 180,E1 -21226.239,E2 -21226.239} C_VEL
LIN {X 0,Y 207.038,Z 314.697,A -85,B 0,C 180,E1 -21230.227,E2 -21230.227} C_VEL
LIN {X 0,Y 207.021,Z 314.693,A -85,B 0,C 180,E1 -21234.154,E2 -21234.154} C_VEL
LIN {X 0,Y 207.345,Z 314.655,A -85,B 0,C 180,E1 -21238.057,E2 -21238.057} C_VEL
LIN {X 0,Y 207.471,Z 314.639,A -85,B 0,C 180,E1 -21239.999,E2 -21239.999} C_VEL
LIN {X 0,Y 207.34,Z 314.652,A -85,B 0,C 180,E1 -21241.941,E2 -21241.941} C_VEL
LIN {X 0,Y 207.1,Z 314.686,A -85,B 0,C 180,E1 -21247.8,E2 -21247.8} C_VEL
LIN {X 0,Y 206.88,Z 314.712,A -85,B 0,C 180,E1 -21251.76,E2 -21251.76} C_VEL
LIN {X 0,Y 206.817,Z 314.724,A -85,B 0,C 180,E1 -21255.774,E2 -21255.774} C_VEL
LIN {X 0,Y 206.725,Z 314.732,A -85,B 0,C 180,E1 -21259.874,E2 -21259.874} C_VEL
LIN {X 0,Y 206.708,Z 314.736,A -85,B 0,C 180,E1 -21264.078,E2 -21264.078} C_VEL
LIN {X 0,Y 206.69,Z 314.737,A -85,B 0,C 180,E1 -21268.426,E2 -21268.426} C_VEL
LIN {X 0,Y 206.664,Z 314.743,A -85,B 0,C 180,E1 -21272.963,E2 -21272.963} C_VEL
LIN {X 0,Y 206.641,Z 314.744,A -85,B 0,C 180,E1 -21277.747,E2 -21277.747} C_VEL
LIN {X 0,Y 206.61,Z 314.749,A -85,B 0,C 180,E1 -21281.565,E2 -21281.565} C_VEL
LIN {X 0,Y 206.608,Z 314.75,A -85,B 0,C 180,E1 -21285.588,E2 -21285.588} C_VEL
LIN {X 0,Y 206.726,Z 314.888,A -85,B 0,C 180,E1 -21291.03,E2 -21291.03} C_VEL
LIN {X 0,Y 209.331,Z 326.58,A -85,B 0,C 180,E1 -21295.644,E2 -21295.644} C_VEL
LIN {X 0,Y 211.861,Z 338.712,A -85,B 0,C 180,E1 -21300.167,E2 -21300.167} C_VEL
LIN {X 0,Y 212.501,Z 341.986,A -85,B 0,C 180,E1 -21301.351,E2 -21301.351} C_VEL
LIN {X 0,Y 212.327,Z 343.693,A -85,B 0,C 180,E1 -21301.932,E2 -21301.932} C_VEL
LIN {X 0,Y 212.447,Z 350.36,A -85,B 0,C 180,E1 -21302.275,E2 -21302.275} C_VEL
LIN {X 0,Y 212.124,Z 356.181,A -85,B 0,C 180,E1 -21302.534,E2 -21302.534} C_VEL
LIN {X 0,Y 207.898,Z 375.369,A -85,B 0,C 180,E1 -21303.22,E2 -21303.22} C_VEL
LIN {X 0,Y 207.666,Z 381.182,A -85,B 0,C 180,E1 -21303.491,E2 -21303.491} C_VEL
LIN {X 0,Y 205.284,Z 442.885,A -85,B 0,C 180,E1 -21306.421,E2 -21306.421} C_VEL
LIN {X 0,Y 204.712,Z 452.606,A -85,B 0,C 180,E1 -21307.087,E2 -21307.087} C_VEL
LIN {X 0,Y 203.898,Z 462.375,A -85,B 0,C 180,E1 -21307.992,E2 -21307.992} C_VEL
LIN {X 0,Y 203.086,Z 470.851,A -85,B 0,C 180,E1 -21308.986,E2 -21308.986} C_VEL
LIN {X 0,Y 202.112,Z 480.812,A -85,B 0,C 180,E1 -21310.453,E2 -21310.453} C_VEL
LIN {X 0,Y 201.193,Z 489.127,A -85,B 0,C 180,E1 -21311.946,E2 -21311.946} C_VEL
LIN {X 0,Y 200.224,Z 497.252,A -85,B 0,C 180,E1 -21313.698,E2 -21313.698} C_VEL
LIN {X 0,Y 199.385,Z 505.068,A -85,B 0,C 180,E1 -21315.721,E2 -21315.721} C_VEL
LIN {X 0,Y 198.786,Z 511.703,A -85,B 0,C 180,E1 -21317.758,E2 -21317.758} C_VEL
LIN {X 0,Y 198.321,Z 518.575,A -85,B 0,C 180,E1 -21320.315,E2 -21320.315} C_VEL
LIN {X 0,Y 198.08,Z 524.204,A -85,B 0,C 180,E1 -21322.872,E2 -21322.872} C_VEL
LIN {X 0,Y 198.027,Z 527.995,A -85,B 0,C 180,E1 -21324.914,E2 -21324.914} C_VEL
LIN {X 0,Y 197.99,Z 532.385,A -85,B 0,C 180,E1 -21327.97,E2 -21327.97} C_VEL
LIN {X 0,Y 198.142,Z 534.621,A -85,B 0,C 180,E1 -21330.004,E2 -21330.004} C_VEL
LIN {X 0,Y 197.616,Z 537.537,A -85,B 0,C 180,E1 -21334.082,E2 -21334.082} C_VEL
LIN {X 0,Y 197.5,Z 538.295,A -85,B 0,C 180,E1 -21336.132,E2 -21336.132} C_VEL
LIN {X 0,Y 197.934,Z 538.714,A -85,B 0,C 180,E1 -21340.229,E2 -21340.229} C_VEL
LIN {X 0,Y 199.303,Z 537.398,A -85,B 0,C 180,E1 -21344.293,E2 -21344.293} C_VEL
LIN {X 0,Y 200.495,Z 536.256,A -85,B 0,C 180,E1 -21346.288,E2 -21346.288} C_VEL
LIN {X 0,Y 202.789,Z 533.651,A -85,B 0,C 180,E1 -21349.225,E2 -21349.225} C_VEL
LIN {X 0,Y 206.373,Z 528.727,A -85,B 0,C 180,E1 -21352.951,E2 -21352.951} C_VEL
LIN {X 0,Y 210.086,Z 523.555,A -85,B 0,C 180,E1 -21355.78,E2 -21355.78} C_VEL
LIN {X 0,Y 213.563,Z 518.438,A -85,B 0,C 180,E1 -21357.967,E2 -21357.967} C_VEL
LIN {X 0,Y 217.388,Z 512.297,A -85,B 0,C 180,E1 -21360.074,E2 -21360.074} C_VEL
LIN {X 0,Y 221.602,Z 504.924,A -85,B 0,C 180,E1 -21362.088,E2 -21362.088} C_VEL
LIN {X 0,Y 225.286,Z 498.049,A -85,B 0,C 180,E1 -21363.624,E2 -21363.624} C_VEL
LIN {X 0,Y 229.587,Z 488.821,A -85,B 0,C 180,E1 -21365.296,E2 -21365.296} C_VEL
LIN {X 0,Y 233.158,Z 480.215,A -85,B 0,C 180,E1 -21366.535,E2 -21366.535} C_VEL
LIN {X 0,Y 236.294,Z 471.446,A -85,B 0,C 180,E1 -21367.569,E2 -21367.569} C_VEL
LIN {X 0,Y 239.671,Z 460.524,A -85,B 0,C 180,E1 -21368.544,E2 -21368.544} C_VEL
LIN {X 0,Y 242.282,Z 450.177,A -85,B 0,C 180,E1 -21369.251,E2 -21369.251} C_VEL
LIN {X 0,Y 244.401,Z 439.106,A -85,B 0,C 180,E1 -21369.804,E2 -21369.804} C_VEL
LIN {X 0,Y 250.088,Z 396.095,A -85,B 0,C 180,E1 -21371.583,E2 -21371.583} C_VEL
LIN {X 0,Y 248.216,Z 390.874,A -85,B 0,C 180,E1 -21373.099,E2 -21373.099} C_VEL
LIN {X 0,Y 245.901,Z 385.326,A -85,B 0,C 180,E1 -21375.139,E2 -21375.139} C_VEL
LIN {X 0,Y 243.276,Z 379.872,A -85,B 0,C 180,E1 -21377.968,E2 -21377.968} C_VEL
LIN {X 0,Y 240.924,Z 375.216,A -85,B 0,C 180,E1 -21381.855,E2 -21381.855} C_VEL
LIN {X 0,Y 240.125,Z 373.886,A -85,B 0,C 180,E1 -21384.172,E2 -21384.172} C_VEL
LIN {X 0,Y 239.963,Z 373.663,A -85,B 0,C 180,E1 -21388.186,E2 -21388.186} C_VEL
LIN {X 0,Y 241.004,Z 374.837,A -85,B 0,C 180,E1 -21391.418,E2 -21391.418} C_VEL
LIN {X 0,Y 243.478,Z 379.382,A -85,B 0,C 180,E1 -21395.439,E2 -21395.439} C_VEL
LIN {X 0,Y 246.115,Z 384.681,A -85,B 0,C 180,E1 -21398.266,E2 -21398.266} C_VEL
LIN {X 0,Y 248.111,Z 389.169,A -85,B 0,C 180,E1 -21400.019,E2 -21400.019} C_VEL
LIN {X 0,Y 249.761,Z 393.595,A -85,B 0,C 180,E1 -21401.421,E2 -21401.421} C_VEL
LIN {X 0,Y 249.518,Z 396.57,A -85,B 0,C 180,E1 -21401.637,E2 -21401.637} C_VEL
LIN {X 0,Y 243.752,Z 435.35,A -85,B 0,C 180,E1 -21403.392,E2 -21403.392} C_VEL
LIN {X 0,Y 240.919,Z 448.527,A -85,B 0,C 180,E1 -21404.286,E2 -21404.286} C_VEL
LIN {X 0,Y 238.058,Z 458.633,A -85,B 0,C 180,E1 -21405.249,E2 -21405.249} C_VEL
LIN {X 0,Y 234.375,Z 469.339,A -85,B 0,C 180,E1 -21406.563,E2 -21406.563} C_VEL
LIN {X 0,Y 231.383,Z 476.896,A -85,B 0,C 180,E1 -21407.725,E2 -21407.725} C_VEL
LIN {X 0,Y 227.545,Z 485.347,A -85,B 0,C 180,E1 -21409.321,E2 -21409.321} C_VEL
LIN {X 0,Y 222.944,Z 494.046,A -85,B 0,C 180,E1 -21411.389,E2 -21411.389} C_VEL
LIN {X 0,Y 218.648,Z 501.073,A -85,B 0,C 180,E1 -21413.605,E2 -21413.605} C_VEL
LIN {X 0,Y 215.658,Z 505.536,A -85,B 0,C 180,E1 -21415.328,E2 -21415.328} C_VEL
LIN {X 0,Y 211.348,Z 510.969,A -85,B 0,C 180,E1 -21418.095,E2 -21418.095} C_VEL
LIN {X 0,Y 208.865,Z 513.833,A -85,B 0,C 180,E1 -21420.001,E2 -21420.001} C_VEL
LIN {X 0,Y 206.593,Z 516.076,A -85,B 0,C 180,E1 -21421.951,E2 -21421.951} C_VEL
LIN {X 0,Y 204.358,Z 517.892,A -85,B 0,C 180,E1 -21424.212,E2 -21424.212} C_VEL
LIN {X 0,Y 201.325,Z 519.451,A -85,B 0,C 180,E1 -21428.028,E2 -21428.028} C_VEL
LIN {X 0,Y 199.986,Z 519.548,A -85,B 0,C 180,E1 -21430.275,E2 -21430.275} C_VEL
LIN {X 0,Y 199.078,Z 519.043,A -85,B 0,C 180,E1 -21432.23,E2 -21432.23} C_VEL
LIN {X 0,Y 198.271,Z 518.04,A -85,B 0,C 180,E1 -21434.368,E2 -21434.368} C_VEL
LIN {X 0,Y 197.532,Z 515.518,A -85,B 0,C 180,E1 -21437.604,E2 -21437.604} C_VEL
LIN {X 0,Y 197.334,Z 511.701,A -85,B 0,C 180,E1 -21440.865,E2 -21440.865} C_VEL
LIN {X 0,Y 197.555,Z 506.296,A -85,B 0,C 180,E1 -21444.15,E2 -21444.15} C_VEL
LIN {X 0,Y 197.993,Z 500.295,A -85,B 0,C 180,E1 -21446.91,E2 -21446.91} C_VEL
LIN {X 0,Y 198.481,Z 494.548,A -85,B 0,C 180,E1 -21449.078,E2 -21449.078} C_VEL
LIN {X 0,Y 199.146,Z 487.193,A -85,B 0,C 180,E1 -21451.37,E2 -21451.37} C_VEL
LIN {X 0,Y 199.976,Z 479.395,A -85,B 0,C 180,E1 -21453.378,E2 -21453.378} C_VEL
LIN {X 0,Y 200.842,Z 470.506,A -85,B 0,C 180,E1 -21455.268,E2 -21455.268} C_VEL
LIN {X 0,Y 201.947,Z 459.109,A -85,B 0,C 180,E1 -21457.203,E2 -21457.203} C_VEL
LIN {X 0,Y 202.816,Z 448.38,A -85,B 0,C 180,E1 -21458.591,E2 -21458.591} C_VEL
LIN {X 0,Y 203.544,Z 438.064,A -85,B 0,C 180,E1 -21459.621,E2 -21459.621} C_VEL
LIN {X 0,Y 204.211,Z 426.324,A -85,B 0,C 180,E1 -21460.472,E2 -21460.472} C_VEL
LIN {X 0,Y 206.466,Z 377.146,A -85,B 0,C 180,E1 -21463.041,E2 -21463.041} C_VEL
LIN {X 0,Y 203.265,Z 342.188,A -85,B 0,C 180,E1 -21465.107,E2 -21465.107} C_VEL
LIN {X 0,Y 203.274,Z 340.737,A -85,B 0,C 180,E1 -21465.256,E2 -21465.256} C_VEL
LIN {X 0,Y 203.8,Z 337.757,A -85,B 0,C 180,E1 -21466.402,E2 -21466.402} C_VEL
LIN {X 0,Y 203.26,Z 333.179,A -85,B 0,C 180,E1 -21468.274,E2 -21468.274} C_VEL
LIN {X 0,Y 201.136,Z 322.378,A -85,B 0,C 180,E1 -21472.933,E2 -21472.933} C_VEL
LIN {X 0,Y 199.69,Z 315.609,A -85,B 0,C 180,E1 -21475.994,E2 -21475.994} C_VEL
LIN {X 0,Y 199.608,Z 315.621,A -85,B 0,C 180,E1 -21480.466,E2 -21480.466} C_VEL
LIN {X 0,Y 199.624,Z 315.618,A -85,B 0,C 180,E1 -21485.007,E2 -21485.007} C_VEL
LIN {X 0,Y 199.653,Z 315.614,A -85,B 0,C 180,E1 -21489.387,E2 -21489.387} C_VEL
LIN {X 0,Y 199.762,Z 315.599,A -85,B 0,C 180,E1 -21493.65,E2 -21493.65} C_VEL
LIN {X 0,Y 199.867,Z 315.585,A -85,B 0,C 180,E1 -21497.817,E2 -21497.817} C_VEL
LIN {X 0,Y 200.079,Z 315.56,A -85,B 0,C 180,E1 -21501.92,E2 -21501.92} C_VEL
LIN {X 0,Y 200.287,Z 315.536,A -85,B 0,C 180,E1 -21507.985,E2 -21507.985} C_VEL
LIN {X 0,Y 200.451,Z 315.516,A -85,B 0,C 180,E1 -21509.996,E2 -21509.996} C_VEL
LIN {X 0,Y 199.987,Z 315.571,A -85,B 0,C 180,E1 -21514.026,E2 -21514.026} C_VEL
LIN {X 0,Y 200.078,Z 315.563,A -85,B 0,C 180,E1 -21518.072,E2 -21518.072} C_VEL
LIN {X 0,Y 199.869,Z 315.586,A -85,B 0,C 180,E1 -21522.174,E2 -21522.174} C_VEL
LIN {X 0,Y 199.763,Z 315.601,A -85,B 0,C 180,E1 -21526.341,E2 -21526.341} C_VEL
LIN {X 0,Y 199.644,Z 315.615,A -85,B 0,C 180,E1 -21530.605,E2 -21530.605} C_VEL
LIN {X 0,Y 199.642,Z 315.616,A -85,B 0,C 180,E1 -21534.981,E2 -21534.981} C_VEL
LIN {X 0,Y 199.599,Z 315.619,A -85,B 0,C 180,E1 -21539.527,E2 -21539.527} C_VEL
LIN {X 0,Y 199.655,Z 315.612,A -85,B 0,C 180,E1 -21542.345,E2 -21542.345} C_VEL
LIN {X 0,Y 199.604,Z 315.618,A -85,B 0,C 180,E1 -21546.758,E2 -21546.758} C_VEL
LIN {X 0,Y 199.581,Z 315.619,A -85,B 0,C 180,E1 -21549.325,E2 -21549.325} C_VEL
LIN {X 0,Y 199.553,Z 315.629,A -85,B 0,C 180,E1 -21552.302,E2 -21552.302} C_VEL
LIN {X 0,Y 199.559,Z 315.625,A -85,B 0,C 180,E1 -21555.221,E2 -21555.221} C_VEL
LIN {X 0,Y 199.553,Z 315.624,A -85,B 0,C 180,E1 -21557.997,E2 -21557.997} C_VEL
LIN {X 0,Y 199.576,Z 315.625,A -85,B 0,C 180,E1 -21560.766,E2 -21560.766} C_VEL
LIN {X 0,Y 199.587,Z 315.619,A -85,B 0,C 180,E1 -21565.707,E2 -21565.707} C_VEL
LIN {X 0,Y 199.667,Z 315.608,A -85,B 0,C 180,E1 -21568.13,E2 -21568.13} C_VEL
LIN {X 0,Y 199.658,Z 315.613,A -85,B 0,C 180,E1 -21572.766,E2 -21572.766} C_VEL
